# B&R Automation Studio project TrakFramework
Automation Studio 4.11.1.147; technology packages: mapp 5.18.0, mappFramework 1.0.0, mappMotion 5.18.0, mappView 5.18.0

## Configuration Config1

CPU PC_any, AutomationRuntime B4.92, Build 4.1.2, Safety 0.0, Vc V4.72.0

### Task classes (Cpu.sw)
```
Cyclic#1 (cycle 400 us, tolerance 0 us):
  AssemblyCt <- Source.AssemblyCtrl.prg
Cyclic#2 (cycle 2400 us, tolerance 2400 us):
  Deciders <- Source.Stations.Deciders.prg
Cyclic#3 (cycle 24000 us, tolerance 48000 us):
  Main <- Source.Main.prg
Cyclic#8 (cycle 800 us):
  Vis <- Source.Vis.Vis.prg
DataObjects: McAcpSys
NcDataObjects: McDriveLog
Binaries: mvLoader, FWRules, McAcpDrv, arsvcreg, McAcpSim, udbdef, TCData, arflatprv, arcoal, Config_3, arconfig, User, Role, sysconf, iomap, asfw, ashwac, ashwd, Config_2, Config_1, Config_4
Libraries: McBase, McAxis, McAcpTrak, standard, AsBrStr, TrakHelper, MpBase, ProcLogic, powerlnk, astime, arssl, fileio, runtime, asieccon, sys_lib
```

### Hardware
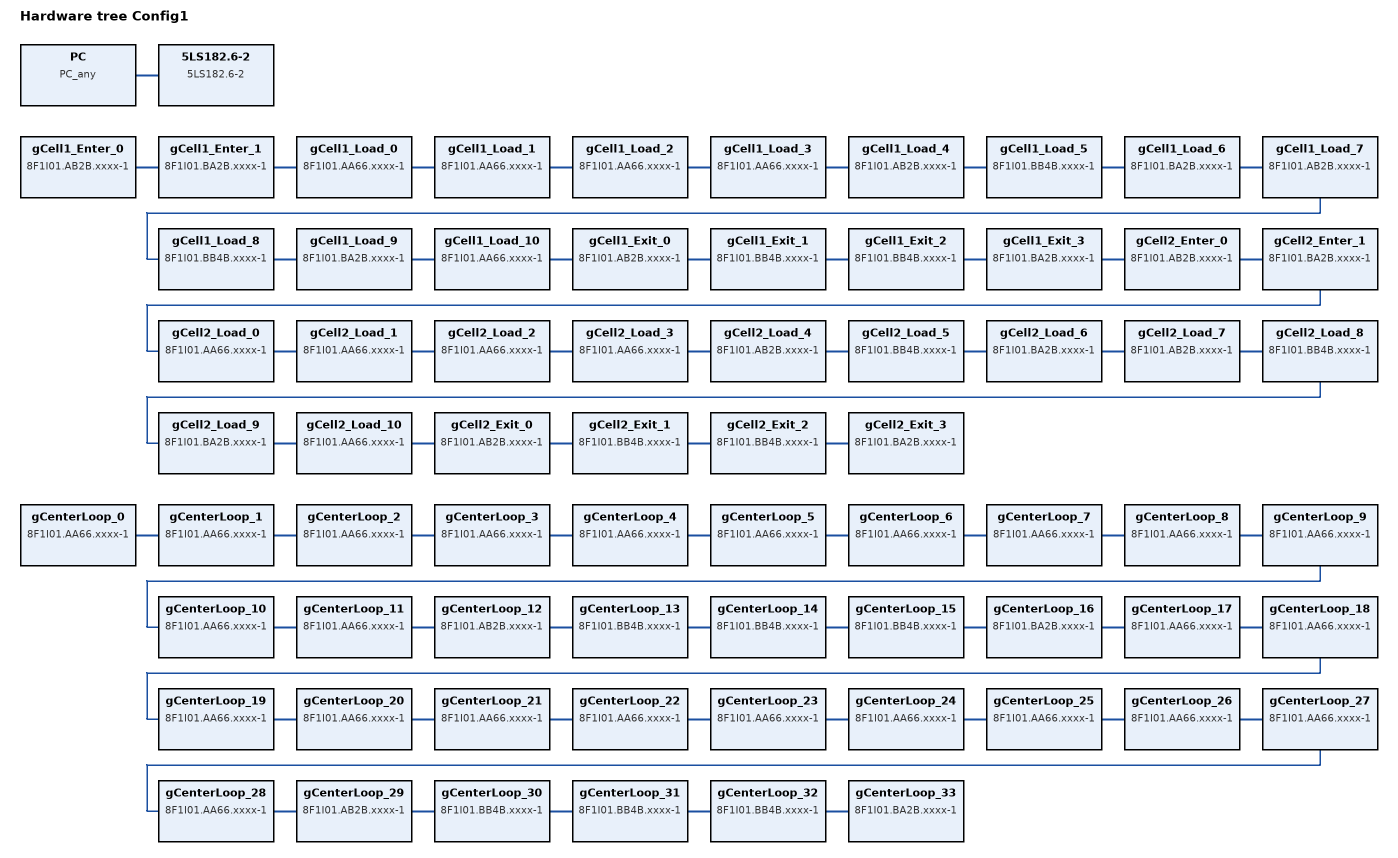
```
5LS182.6-2 : 5LS182.6-2 v1.9.0.0  [SL -> PC.SL1]
  Connector IF1:
    DNAConfiguration = manual
PC : PC_any v1.1.1.0 (OrderNumber=PC)
  ConfigurationID = BundlingSim_Config1
  SystemTick = 400
  Cyclic1Duration = 400
  Cyclic1Tolerance = 0
  Cyclic2Duration = 2400
  Cyclic2Tolerance = 2400
  Cyclic3Duration = 24000
  Cyclic3Tolerance = 48000
  Cyclic8Duration = 800
  FileDevice1
  FileDeviceName1 = SvgData
  FileDevicePath1 = ../../../../Logical/Scene
  ActivateOpcUa = 1
  OpcUaInformationModels_PV_Version = 1
gCell1_Enter_0 : 8F1I01.AB2B.xxxx-1 v1.0.0.2  [PLK1 -> gCenterLoop_33.PLK2 [Cable Type=PowerlinkCable, Length=10, Version=1.0.0.3]; PLK2 -> gCell1_Enter_1.PLK1 [Cable Type=PowerlinkCable, Length=10, Version=1.0.0.3]]
  DriveConfiguration:
    McTypeID = LLMConfig
  DriveConfiguration/Segment:
    Shape = STRAIGHT105_TO_CIRCULAR
    SegmentReference = gCell1_Enter_0
    StopReaction = UseAssemblySetting
    SpeedFilter = UseAssemblySetting
gCell1_Enter_1 : 8F1I01.BA2B.xxxx-1 v1.0.0.2  [PLK1 -> gCell1_Enter_0.PLK2 [Cable Type=PowerlinkCable, Length=10, Version=1.0.0.3]; PLK2 -> gCell1_Load_0.PLK1 [Cable Type=PowerlinkCable, Length=10, Version=1.0.0.3]]
  DriveConfiguration:
    McTypeID = LLMConfig
  DriveConfiguration/Segment:
    Shape = CIRCULAR_TO_STRAIGHT105
    SegmentReference = gCell1_Enter_1
    StopReaction = UseAssemblySetting
    SpeedFilter = UseAssemblySetting
gCell1_Exit_0 : 8F1I01.AB2B.xxxx-1 v1.0.0.2  [PLK1 -> gCell1_Load_10.PLK2 [Cable Type=PowerlinkCable, Length=10, Version=1.0.0.3]; PLK2 -> gCell1_Exit_1.PLK1 [Cable Type=PowerlinkCable, Length=10, Version=1.0.0.3]]
  DriveConfiguration:
    McTypeID = LLMConfig
  DriveConfiguration/Segment:
    Shape = STRAIGHT105_TO_CIRCULAR
    SegmentReference = gCell1_Exit_0
    StopReaction = UseAssemblySetting
    SpeedFilter = UseAssemblySetting
gCell1_Exit_1 : 8F1I01.BB4B.xxxx-1 v1.0.0.2  [PLK1 -> gCell1_Exit_0.PLK2 [Cable Type=PowerlinkCable, Length=10, Version=1.0.0.3]; PLK2 -> gCell1_Exit_2.PLK1 [Cable Type=PowerlinkCable, Length=10, Version=1.0.0.3]]
  DriveConfiguration:
    McTypeID = LLMConfig
  DriveConfiguration/Segment:
    Shape = CIRCULAR
    SegmentReference = gCell1_Exit_1
    StopReaction = UseAssemblySetting
    SpeedFilter = UseAssemblySetting
gCell1_Exit_2 : 8F1I01.BB4B.xxxx-1 v1.0.0.2  [PLK1 -> gCell1_Exit_1.PLK2 [Cable Type=PowerlinkCable, Length=10, Version=1.0.0.3]; PLK2 -> gCell1_Exit_3.PLK1 [Cable Type=PowerlinkCable, Length=10, Version=1.0.0.3]]
  DriveConfiguration:
    McTypeID = LLMConfig
  DriveConfiguration/Segment:
    Shape = CIRCULAR
    SegmentReference = gCell1_Exit_2
    StopReaction = UseAssemblySetting
    SpeedFilter = UseAssemblySetting
gCell1_Exit_3 : 8F1I01.BA2B.xxxx-1 v1.0.0.2  [PLK1 -> gCell1_Exit_2.PLK2 [Cable Type=PowerlinkCable, Length=10, Version=1.0.0.3]; PLK2 -> gCell2_Enter_0.PLK1 [Cable Type=PowerlinkCable, Length=10, Version=1.0.0.3]]
  DriveConfiguration:
    McTypeID = LLMConfig
  DriveConfiguration/Segment:
    Shape = CIRCULAR_TO_STRAIGHT105
    SegmentReference = gCell1_Exit_3
    StopReaction = UseAssemblySetting
    SpeedFilter = UseAssemblySetting
gCell1_Load_0 : 8F1I01.AA66.xxxx-1 v1.0.0.2  [PLK1 -> gCell1_Enter_1.PLK2 [Cable Type=PowerlinkCable, Length=10, Version=1.0.0.3]; PLK2 -> gCell1_Load_1.PLK1 [Cable Type=PowerlinkCable, Length=10, Version=1.0.0.3]]
  DriveConfiguration:
    McTypeID = LLMConfig
  DriveConfiguration/Segment:
    Shape = STRAIGHT660
    SegmentReference = gCell1_Load_0
    StopReaction = UseAssemblySetting
    SpeedFilter = UseAssemblySetting
gCell1_Load_1 : 8F1I01.AA66.xxxx-1 v1.0.0.2  [PLK1 -> gCell1_Load_0.PLK2 [Cable Type=PowerlinkCable, Length=10, Version=1.0.0.3]; PLK2 -> gCell1_Load_2.PLK1 [Cable Type=PowerlinkCable, Length=10, Version=1.0.0.3]]
  DriveConfiguration:
    McTypeID = LLMConfig
  DriveConfiguration/Segment:
    Shape = STRAIGHT660
    SegmentReference = gCell1_Load_1
    StopReaction = UseAssemblySetting
    SpeedFilter = UseAssemblySetting
gCell1_Load_10 : 8F1I01.AA66.xxxx-1 v1.0.0.2  [PLK1 -> gCell1_Load_9.PLK2 [Cable Type=PowerlinkCable, Length=10, Version=1.0.0.3]; PLK2 -> gCell1_Exit_0.PLK1 [Cable Type=PowerlinkCable, Length=10, Version=1.0.0.3]]
  DriveConfiguration:
    McTypeID = LLMConfig
  DriveConfiguration/Segment:
    Shape = STRAIGHT660
    SegmentReference = gCell1_Load_10
    StopReaction = UseAssemblySetting
    SpeedFilter = UseAssemblySetting
gCell1_Load_2 : 8F1I01.AA66.xxxx-1 v1.0.0.2  [PLK1 -> gCell1_Load_1.PLK2 [Cable Type=PowerlinkCable, Length=10, Version=1.0.0.3]; PLK2 -> gCell1_Load_3.PLK1 [Cable Type=PowerlinkCable, Length=10, Version=1.0.0.3]]
  DriveConfiguration:
    McTypeID = LLMConfig
  DriveConfiguration/Segment:
    Shape = STRAIGHT660
    SegmentReference = gCell1_Load_2
    StopReaction = UseAssemblySetting
    SpeedFilter = UseAssemblySetting
gCell1_Load_3 : 8F1I01.AA66.xxxx-1 v1.0.0.2  [PLK1 -> gCell1_Load_2.PLK2 [Cable Type=PowerlinkCable, Length=10, Version=1.0.0.3]; PLK2 -> gCell1_Load_4.PLK1 [Cable Type=PowerlinkCable, Length=10, Version=1.0.0.3]]
  DriveConfiguration:
    McTypeID = LLMConfig
  DriveConfiguration/Segment:
    Shape = STRAIGHT660
    SegmentReference = gCell1_Load_3
    StopReaction = UseAssemblySetting
    SpeedFilter = UseAssemblySetting
gCell1_Load_4 : 8F1I01.AB2B.xxxx-1 v1.0.0.2  [PLK1 -> gCell1_Load_3.PLK2 [Cable Type=PowerlinkCable, Length=10, Version=1.0.0.3]; PLK2 -> gCell1_Load_5.PLK1 [Cable Type=PowerlinkCable, Length=10, Version=1.0.0.3]]
  DriveConfiguration:
    McTypeID = LLMConfig
  DriveConfiguration/Segment:
    Shape = STRAIGHT105_TO_CIRCULAR
    SegmentReference = gCell1_Load_4
    StopReaction = UseAssemblySetting
    SpeedFilter = UseAssemblySetting
gCell1_Load_5 : 8F1I01.BB4B.xxxx-1 v1.0.0.2  [PLK1 -> gCell1_Load_4.PLK2 [Cable Type=PowerlinkCable, Length=10, Version=1.0.0.3]; PLK2 -> gCell1_Load_6.PLK1 [Cable Type=PowerlinkCable, Length=10, Version=1.0.0.3]]
  DriveConfiguration:
    McTypeID = LLMConfig
  DriveConfiguration/Segment:
    Shape = CIRCULAR
    SegmentReference = gCell1_Load_5
    StopReaction = UseAssemblySetting
    SpeedFilter = UseAssemblySetting
gCell1_Load_6 : 8F1I01.BA2B.xxxx-1 v1.0.0.2  [PLK1 -> gCell1_Load_5.PLK2 [Cable Type=PowerlinkCable, Length=10, Version=1.0.0.3]; PLK2 -> gCell1_Load_7.PLK1 [Cable Type=PowerlinkCable, Length=10, Version=1.0.0.3]]
  DriveConfiguration:
    McTypeID = LLMConfig
  DriveConfiguration/Segment:
    Shape = CIRCULAR_TO_STRAIGHT105
    SegmentReference = gCell1_Load_6
    StopReaction = UseAssemblySetting
    SpeedFilter = UseAssemblySetting
gCell1_Load_7 : 8F1I01.AB2B.xxxx-1 v1.0.0.2  [PLK1 -> gCell1_Load_6.PLK2 [Cable Type=PowerlinkCable, Length=10, Version=1.0.0.3]; PLK2 -> gCell1_Load_8.PLK1 [Cable Type=PowerlinkCable, Length=10, Version=1.0.0.3]]
  DriveConfiguration:
    McTypeID = LLMConfig
  DriveConfiguration/Segment:
    Shape = STRAIGHT105_TO_CIRCULAR
    SegmentReference = gCell1_Load_7
    StopReaction = UseAssemblySetting
    SpeedFilter = UseAssemblySetting
gCell1_Load_8 : 8F1I01.BB4B.xxxx-1 v1.0.0.2  [PLK1 -> gCell1_Load_7.PLK2 [Cable Type=PowerlinkCable, Length=10, Version=1.0.0.3]; PLK2 -> gCell1_Load_9.PLK1 [Cable Type=PowerlinkCable, Length=10, Version=1.0.0.3]]
  DriveConfiguration:
    McTypeID = LLMConfig
  DriveConfiguration/Segment:
    Shape = CIRCULAR
    SegmentReference = gCell1_Load_8
    StopReaction = UseAssemblySetting
    SpeedFilter = UseAssemblySetting
gCell1_Load_9 : 8F1I01.BA2B.xxxx-1 v1.0.0.2  [PLK1 -> gCell1_Load_8.PLK2 [Cable Type=PowerlinkCable, Length=10, Version=1.0.0.3]; PLK2 -> gCell1_Load_10.PLK1 [Cable Type=PowerlinkCable, Length=10, Version=1.0.0.3]]
  DriveConfiguration:
    McTypeID = LLMConfig
  DriveConfiguration/Segment:
    Shape = CIRCULAR_TO_STRAIGHT105
    SegmentReference = gCell1_Load_9
    StopReaction = UseAssemblySetting
    SpeedFilter = UseAssemblySetting
gCell2_Enter_0 : 8F1I01.AB2B.xxxx-1 v1.0.0.2  [PLK1 -> gCell1_Exit_3.PLK2 [Cable Type=PowerlinkCable, Length=10, Version=1.0.0.3]; PLK2 -> gCell2_Enter_1.PLK1 [Cable Type=PowerlinkCable, Length=10, Version=1.0.0.3]]
  DriveConfiguration:
    McTypeID = LLMConfig
  DriveConfiguration/Segment:
    Shape = STRAIGHT105_TO_CIRCULAR
    SegmentReference = gCell2_Enter_0
    StopReaction = UseAssemblySetting
    SpeedFilter = UseAssemblySetting
gCell2_Enter_1 : 8F1I01.BA2B.xxxx-1 v1.0.0.2  [PLK1 -> gCell2_Enter_0.PLK2 [Cable Type=PowerlinkCable, Length=10, Version=1.0.0.3]; PLK2 -> gCell2_Load_0.PLK1 [Cable Type=PowerlinkCable, Length=10, Version=1.0.0.3]]
  DriveConfiguration:
    McTypeID = LLMConfig
  DriveConfiguration/Segment:
    Shape = CIRCULAR_TO_STRAIGHT105
    SegmentReference = gCell2_Enter_1
    StopReaction = UseAssemblySetting
    SpeedFilter = UseAssemblySetting
gCell2_Exit_0 : 8F1I01.AB2B.xxxx-1 v1.0.0.2  [PLK1 -> gCell2_Load_10.PLK2 [Cable Type=PowerlinkCable, Length=10, Version=1.0.0.3]; PLK2 -> gCell2_Exit_1.PLK1 [Cable Type=PowerlinkCable, Length=10, Version=1.0.0.3]]
  DriveConfiguration:
    McTypeID = LLMConfig
  DriveConfiguration/Segment:
    Shape = STRAIGHT105_TO_CIRCULAR
    SegmentReference = gCell2_Exit_0
    StopReaction = UseAssemblySetting
    SpeedFilter = UseAssemblySetting
gCell2_Exit_1 : 8F1I01.BB4B.xxxx-1 v1.0.0.2  [PLK1 -> gCell2_Exit_0.PLK2 [Cable Type=PowerlinkCable, Length=10, Version=1.0.0.3]; PLK2 -> gCell2_Exit_2.PLK1 [Cable Type=PowerlinkCable, Length=10, Version=1.0.0.3]]
  DriveConfiguration:
    McTypeID = LLMConfig
  DriveConfiguration/Segment:
    Shape = CIRCULAR
    SegmentReference = gCell2_Exit_1
    StopReaction = UseAssemblySetting
    SpeedFilter = UseAssemblySetting
gCell2_Exit_2 : 8F1I01.BB4B.xxxx-1 v1.0.0.2  [PLK1 -> gCell2_Exit_1.PLK2 [Cable Type=PowerlinkCable, Length=10, Version=1.0.0.3]; PLK2 -> gCell2_Exit_3.PLK1 [Cable Type=PowerlinkCable, Length=10, Version=1.0.0.3]]
  DriveConfiguration:
    McTypeID = LLMConfig
  DriveConfiguration/Segment:
    Shape = CIRCULAR
    SegmentReference = gCell2_Exit_2
    StopReaction = UseAssemblySetting
    SpeedFilter = UseAssemblySetting
gCell2_Exit_3 : 8F1I01.BA2B.xxxx-1 v1.0.0.2  [PLK1 -> gCell2_Exit_2.PLK2 [Cable Type=PowerlinkCable, Length=10, Version=1.0.0.3]]
  DriveConfiguration:
    McTypeID = LLMConfig
  DriveConfiguration/Segment:
    Shape = CIRCULAR_TO_STRAIGHT105
    SegmentReference = gCell2_Exit_3
    StopReaction = UseAssemblySetting
    SpeedFilter = UseAssemblySetting
gCell2_Load_0 : 8F1I01.AA66.xxxx-1 v1.0.0.2  [PLK1 -> gCell2_Enter_1.PLK2 [Cable Type=PowerlinkCable, Length=10, Version=1.0.0.3]; PLK2 -> gCell2_Load_1.PLK1 [Cable Type=PowerlinkCable, Length=10, Version=1.0.0.3]]
  DriveConfiguration:
    McTypeID = LLMConfig
  DriveConfiguration/Segment:
    Shape = STRAIGHT660
    SegmentReference = gCell2_Load_0
    StopReaction = UseAssemblySetting
    SpeedFilter = UseAssemblySetting
gCell2_Load_1 : 8F1I01.AA66.xxxx-1 v1.0.0.2  [PLK1 -> gCell2_Load_0.PLK2 [Cable Type=PowerlinkCable, Length=10, Version=1.0.0.3]; PLK2 -> gCell2_Load_2.PLK1 [Cable Type=PowerlinkCable, Length=10, Version=1.0.0.3]]
  DriveConfiguration:
    McTypeID = LLMConfig
  DriveConfiguration/Segment:
    Shape = STRAIGHT660
    SegmentReference = gCell2_Load_1
    StopReaction = UseAssemblySetting
    SpeedFilter = UseAssemblySetting
gCell2_Load_10 : 8F1I01.AA66.xxxx-1 v1.0.0.2  [PLK1 -> gCell2_Load_9.PLK2 [Cable Type=PowerlinkCable, Length=10, Version=1.0.0.3]; PLK2 -> gCell2_Exit_0.PLK1 [Cable Type=PowerlinkCable, Length=10, Version=1.0.0.3]]
  DriveConfiguration:
    McTypeID = LLMConfig
  DriveConfiguration/Segment:
    Shape = STRAIGHT660
    SegmentReference = gCell2_Load_10
    StopReaction = UseAssemblySetting
    SpeedFilter = UseAssemblySetting
gCell2_Load_2 : 8F1I01.AA66.xxxx-1 v1.0.0.2  [PLK1 -> gCell2_Load_1.PLK2 [Cable Type=PowerlinkCable, Length=10, Version=1.0.0.3]; PLK2 -> gCell2_Load_3.PLK1 [Cable Type=PowerlinkCable, Length=10, Version=1.0.0.3]]
  DriveConfiguration:
    McTypeID = LLMConfig
  DriveConfiguration/Segment:
    Shape = STRAIGHT660
    SegmentReference = gCell2_Load_2
    StopReaction = UseAssemblySetting
    SpeedFilter = UseAssemblySetting
gCell2_Load_3 : 8F1I01.AA66.xxxx-1 v1.0.0.2  [PLK1 -> gCell2_Load_2.PLK2 [Cable Type=PowerlinkCable, Length=10, Version=1.0.0.3]; PLK2 -> gCell2_Load_4.PLK1 [Cable Type=PowerlinkCable, Length=10, Version=1.0.0.3]]
  DriveConfiguration:
    McTypeID = LLMConfig
  DriveConfiguration/Segment:
    Shape = STRAIGHT660
    SegmentReference = gCell2_Load_3
    StopReaction = UseAssemblySetting
    SpeedFilter = UseAssemblySetting
gCell2_Load_4 : 8F1I01.AB2B.xxxx-1 v1.0.0.2  [PLK1 -> gCell2_Load_3.PLK2 [Cable Type=PowerlinkCable, Length=10, Version=1.0.0.3]; PLK2 -> gCell2_Load_5.PLK1 [Cable Type=PowerlinkCable, Length=10, Version=1.0.0.3]]
  DriveConfiguration:
    McTypeID = LLMConfig
  DriveConfiguration/Segment:
    Shape = STRAIGHT105_TO_CIRCULAR
    SegmentReference = gCell2_Load_4
    StopReaction = UseAssemblySetting
    SpeedFilter = UseAssemblySetting
gCell2_Load_5 : 8F1I01.BB4B.xxxx-1 v1.0.0.2  [PLK1 -> gCell2_Load_4.PLK2 [Cable Type=PowerlinkCable, Length=10, Version=1.0.0.3]; PLK2 -> gCell2_Load_6.PLK1 [Cable Type=PowerlinkCable, Length=10, Version=1.0.0.3]]
  DriveConfiguration:
    McTypeID = LLMConfig
  DriveConfiguration/Segment:
    Shape = CIRCULAR
    SegmentReference = gCell2_Load_5
    StopReaction = UseAssemblySetting
    SpeedFilter = UseAssemblySetting
gCell2_Load_6 : 8F1I01.BA2B.xxxx-1 v1.0.0.2  [PLK1 -> gCell2_Load_5.PLK2 [Cable Type=PowerlinkCable, Length=10, Version=1.0.0.3]; PLK2 -> gCell2_Load_7.PLK1 [Cable Type=PowerlinkCable, Length=10, Version=1.0.0.3]]
  DriveConfiguration:
    McTypeID = LLMConfig
  DriveConfiguration/Segment:
    Shape = CIRCULAR_TO_STRAIGHT105
    SegmentReference = gCell2_Load_6
    StopReaction = UseAssemblySetting
    SpeedFilter = UseAssemblySetting
gCell2_Load_7 : 8F1I01.AB2B.xxxx-1 v1.0.0.2  [PLK1 -> gCell2_Load_6.PLK2 [Cable Type=PowerlinkCable, Length=10, Version=1.0.0.3]; PLK2 -> gCell2_Load_8.PLK1 [Cable Type=PowerlinkCable, Length=10, Version=1.0.0.3]]
  DriveConfiguration:
    McTypeID = LLMConfig
  DriveConfiguration/Segment:
    Shape = STRAIGHT105_TO_CIRCULAR
    SegmentReference = gCell2_Load_7
    StopReaction = UseAssemblySetting
    SpeedFilter = UseAssemblySetting
gCell2_Load_8 : 8F1I01.BB4B.xxxx-1 v1.0.0.2  [PLK1 -> gCell2_Load_7.PLK2 [Cable Type=PowerlinkCable, Length=10, Version=1.0.0.3]; PLK2 -> gCell2_Load_9.PLK1 [Cable Type=PowerlinkCable, Length=10, Version=1.0.0.3]]
  DriveConfiguration:
    McTypeID = LLMConfig
  DriveConfiguration/Segment:
    Shape = CIRCULAR
    SegmentReference = gCell2_Load_8
    StopReaction = UseAssemblySetting
    SpeedFilter = UseAssemblySetting
gCell2_Load_9 : 8F1I01.BA2B.xxxx-1 v1.0.0.2  [PLK1 -> gCell2_Load_8.PLK2 [Cable Type=PowerlinkCable, Length=10, Version=1.0.0.3]; PLK2 -> gCell2_Load_10.PLK1 [Cable Type=PowerlinkCable, Length=10, Version=1.0.0.3]]
  DriveConfiguration:
    McTypeID = LLMConfig
  DriveConfiguration/Segment:
    Shape = CIRCULAR_TO_STRAIGHT105
    SegmentReference = gCell2_Load_9
    StopReaction = UseAssemblySetting
    SpeedFilter = UseAssemblySetting
gCenterLoop_0 : 8F1I01.AA66.xxxx-1 v1.0.0.2  [PLK2 -> gCenterLoop_1.PLK1 [Cable Type=PowerlinkCable, Length=10, Version=1.0.0.3]; PLK3 -> 5LS182.6-2.IF1 [Cable Type=PowerlinkCable, Length=10, Version=1.0.0.3]]
  DriveConfiguration:
    McTypeID = LLMConfig
  DriveConfiguration/Segment:
    Shape = STRAIGHT660
    SegmentReference = gCenterLoop_0
    StopReaction = UseAssemblySetting
    SpeedFilter = UseAssemblySetting
gCenterLoop_1 : 8F1I01.AA66.xxxx-1 v1.0.0.2  [PLK1 -> gCenterLoop_0.PLK2 [Cable Type=PowerlinkCable, Length=10, Version=1.0.0.3]; PLK2 -> gCenterLoop_2.PLK1 [Cable Type=PowerlinkCable, Length=10, Version=1.0.0.3]]
  DriveConfiguration:
    McTypeID = LLMConfig
  DriveConfiguration/Segment:
    Shape = STRAIGHT660
    SegmentReference = gCenterLoop_1
    StopReaction = UseAssemblySetting
    SpeedFilter = UseAssemblySetting
gCenterLoop_10 : 8F1I01.AA66.xxxx-1 v1.0.0.2  [PLK1 -> gCenterLoop_9.PLK2 [Cable Type=PowerlinkCable, Length=10, Version=1.0.0.3]; PLK2 -> gCenterLoop_11.PLK1 [Cable Type=PowerlinkCable, Length=10, Version=1.0.0.3]]
  DriveConfiguration:
    McTypeID = LLMConfig
  DriveConfiguration/Segment:
    Shape = STRAIGHT660
    SegmentReference = gCenterLoop_10
    StopReaction = UseAssemblySetting
    SpeedFilter = UseAssemblySetting
gCenterLoop_11 : 8F1I01.AA66.xxxx-1 v1.0.0.2  [PLK1 -> gCenterLoop_10.PLK2 [Cable Type=PowerlinkCable, Length=10, Version=1.0.0.3]; PLK2 -> gCenterLoop_12.PLK1 [Cable Type=PowerlinkCable, Length=10, Version=1.0.0.3]]
  DriveConfiguration:
    McTypeID = LLMConfig
  DriveConfiguration/Segment:
    Shape = STRAIGHT660
    SegmentReference = gCenterLoop_11
    StopReaction = UseAssemblySetting
    SpeedFilter = UseAssemblySetting
gCenterLoop_12 : 8F1I01.AB2B.xxxx-1 v1.0.0.2  [PLK1 -> gCenterLoop_11.PLK2 [Cable Type=PowerlinkCable, Length=10, Version=1.0.0.3]; PLK2 -> gCenterLoop_13.PLK1 [Cable Type=PowerlinkCable, Length=10, Version=1.0.0.3]]
  DriveConfiguration:
    McTypeID = LLMConfig
  DriveConfiguration/Segment:
    Shape = STRAIGHT105_TO_CIRCULAR
    SegmentReference = gCenterLoop_12
    StopReaction = UseAssemblySetting
    SpeedFilter = UseAssemblySetting
gCenterLoop_13 : 8F1I01.BB4B.xxxx-1 v1.0.0.2  [PLK1 -> gCenterLoop_12.PLK2 [Cable Type=PowerlinkCable, Length=10, Version=1.0.0.3]; PLK2 -> gCenterLoop_14.PLK1 [Cable Type=PowerlinkCable, Length=10, Version=1.0.0.3]]
  DriveConfiguration:
    McTypeID = LLMConfig
  DriveConfiguration/Segment:
    Shape = CIRCULAR
    SegmentReference = gCenterLoop_13
    StopReaction = UseAssemblySetting
    SpeedFilter = UseAssemblySetting
gCenterLoop_14 : 8F1I01.BB4B.xxxx-1 v1.0.0.2  [PLK1 -> gCenterLoop_13.PLK2 [Cable Type=PowerlinkCable, Length=10, Version=1.0.0.3]; PLK2 -> gCenterLoop_15.PLK1 [Cable Type=PowerlinkCable, Length=10, Version=1.0.0.3]]
  DriveConfiguration:
    McTypeID = LLMConfig
  DriveConfiguration/Segment:
    Shape = CIRCULAR
    SegmentReference = gCenterLoop_14
    StopReaction = UseAssemblySetting
    SpeedFilter = UseAssemblySetting
gCenterLoop_15 : 8F1I01.BB4B.xxxx-1 v1.0.0.2  [PLK1 -> gCenterLoop_14.PLK2 [Cable Type=PowerlinkCable, Length=10, Version=1.0.0.3]; PLK2 -> gCenterLoop_16.PLK1 [Cable Type=PowerlinkCable, Length=10, Version=1.0.0.3]]
  DriveConfiguration:
    McTypeID = LLMConfig
  DriveConfiguration/Segment:
    Shape = CIRCULAR
    SegmentReference = gCenterLoop_15
    StopReaction = UseAssemblySetting
    SpeedFilter = UseAssemblySetting
gCenterLoop_16 : 8F1I01.BA2B.xxxx-1 v1.0.0.2  [PLK1 -> gCenterLoop_15.PLK2 [Cable Type=PowerlinkCable, Length=10, Version=1.0.0.3]; PLK2 -> gCenterLoop_17.PLK1 [Cable Type=PowerlinkCable, Length=10, Version=1.0.0.3]]
  DriveConfiguration:
    McTypeID = LLMConfig
  DriveConfiguration/Segment:
    Shape = CIRCULAR_TO_STRAIGHT105
    SegmentReference = gCenterLoop_16
    StopReaction = UseAssemblySetting
    SpeedFilter = UseAssemblySetting
gCenterLoop_17 : 8F1I01.AA66.xxxx-1 v1.0.0.2  [PLK1 -> gCenterLoop_16.PLK2 [Cable Type=PowerlinkCable, Length=10, Version=1.0.0.3]; PLK2 -> gCenterLoop_18.PLK1 [Cable Type=PowerlinkCable, Length=10, Version=1.0.0.3]]
  DriveConfiguration:
    McTypeID = LLMConfig
  DriveConfiguration/Segment:
    Shape = STRAIGHT660
    SegmentReference = gCenterLoop_17
    StopReaction = UseAssemblySetting
    SpeedFilter = UseAssemblySetting
gCenterLoop_18 : 8F1I01.AA66.xxxx-1 v1.0.0.2  [PLK1 -> gCenterLoop_17.PLK2 [Cable Type=PowerlinkCable, Length=10, Version=1.0.0.3]; PLK2 -> gCenterLoop_19.PLK1 [Cable Type=PowerlinkCable, Length=10, Version=1.0.0.3]]
  DriveConfiguration:
    McTypeID = LLMConfig
  DriveConfiguration/Segment:
    Shape = STRAIGHT660
    SegmentReference = gCenterLoop_18
    StopReaction = UseAssemblySetting
    SpeedFilter = UseAssemblySetting
gCenterLoop_19 : 8F1I01.AA66.xxxx-1 v1.0.0.2  [PLK1 -> gCenterLoop_18.PLK2 [Cable Type=PowerlinkCable, Length=10, Version=1.0.0.3]; PLK2 -> gCenterLoop_20.PLK1 [Cable Type=PowerlinkCable, Length=10, Version=1.0.0.3]]
  DriveConfiguration:
    McTypeID = LLMConfig
  DriveConfiguration/Segment:
    Shape = STRAIGHT660
    SegmentReference = gCenterLoop_19
    StopReaction = UseAssemblySetting
    SpeedFilter = UseAssemblySetting
gCenterLoop_2 : 8F1I01.AA66.xxxx-1 v1.0.0.2  [PLK1 -> gCenterLoop_1.PLK2 [Cable Type=PowerlinkCable, Length=10, Version=1.0.0.3]; PLK2 -> gCenterLoop_3.PLK1 [Cable Type=PowerlinkCable, Length=10, Version=1.0.0.3]]
  DriveConfiguration:
    McTypeID = LLMConfig
  DriveConfiguration/Segment:
    Shape = STRAIGHT660
    SegmentReference = gCenterLoop_2
    StopReaction = UseAssemblySetting
    SpeedFilter = UseAssemblySetting
gCenterLoop_20 : 8F1I01.AA66.xxxx-1 v1.0.0.2  [PLK1 -> gCenterLoop_19.PLK2 [Cable Type=PowerlinkCable, Length=10, Version=1.0.0.3]; PLK2 -> gCenterLoop_21.PLK1 [Cable Type=PowerlinkCable, Length=10, Version=1.0.0.3]]
  DriveConfiguration:
    McTypeID = LLMConfig
  DriveConfiguration/Segment:
    Shape = STRAIGHT660
    SegmentReference = gCenterLoop_20
    StopReaction = UseAssemblySetting
    SpeedFilter = UseAssemblySetting
gCenterLoop_21 : 8F1I01.AA66.xxxx-1 v1.0.0.2  [PLK1 -> gCenterLoop_20.PLK2 [Cable Type=PowerlinkCable, Length=10, Version=1.0.0.3]; PLK2 -> gCenterLoop_22.PLK1 [Cable Type=PowerlinkCable, Length=10, Version=1.0.0.3]]
  DriveConfiguration:
    McTypeID = LLMConfig
  DriveConfiguration/Segment:
    Shape = STRAIGHT660
    SegmentReference = gCenterLoop_21
    StopReaction = UseAssemblySetting
    SpeedFilter = UseAssemblySetting
gCenterLoop_22 : 8F1I01.AA66.xxxx-1 v1.0.0.2  [PLK1 -> gCenterLoop_21.PLK2 [Cable Type=PowerlinkCable, Length=10, Version=1.0.0.3]; PLK2 -> gCenterLoop_23.PLK1 [Cable Type=PowerlinkCable, Length=10, Version=1.0.0.3]]
  DriveConfiguration:
    McTypeID = LLMConfig
  DriveConfiguration/Segment:
    Shape = STRAIGHT660
    SegmentReference = gCenterLoop_22
    StopReaction = UseAssemblySetting
    SpeedFilter = UseAssemblySetting
gCenterLoop_23 : 8F1I01.AA66.xxxx-1 v1.0.0.2  [PLK1 -> gCenterLoop_22.PLK2 [Cable Type=PowerlinkCable, Length=10, Version=1.0.0.3]; PLK2 -> gCenterLoop_24.PLK1 [Cable Type=PowerlinkCable, Length=10, Version=1.0.0.3]]
  DriveConfiguration:
    McTypeID = LLMConfig
  DriveConfiguration/Segment:
    Shape = STRAIGHT660
    SegmentReference = gCenterLoop_23
    StopReaction = UseAssemblySetting
    SpeedFilter = UseAssemblySetting
gCenterLoop_24 : 8F1I01.AA66.xxxx-1 v1.0.0.2  [PLK1 -> gCenterLoop_23.PLK2 [Cable Type=PowerlinkCable, Length=10, Version=1.0.0.3]; PLK2 -> gCenterLoop_25.PLK1 [Cable Type=PowerlinkCable, Length=10, Version=1.0.0.3]]
  DriveConfiguration:
    McTypeID = LLMConfig
  DriveConfiguration/Segment:
    Shape = STRAIGHT660
    SegmentReference = gCenterLoop_24
    StopReaction = UseAssemblySetting
    SpeedFilter = UseAssemblySetting
gCenterLoop_25 : 8F1I01.AA66.xxxx-1 v1.0.0.2  [PLK1 -> gCenterLoop_24.PLK2 [Cable Type=PowerlinkCable, Length=10, Version=1.0.0.3]; PLK2 -> gCenterLoop_26.PLK1 [Cable Type=PowerlinkCable, Length=10, Version=1.0.0.3]]
  DriveConfiguration:
    McTypeID = LLMConfig
  DriveConfiguration/Segment:
    Shape = STRAIGHT660
    SegmentReference = gCenterLoop_25
    StopReaction = UseAssemblySetting
    SpeedFilter = UseAssemblySetting
gCenterLoop_26 : 8F1I01.AA66.xxxx-1 v1.0.0.2  [PLK1 -> gCenterLoop_25.PLK2 (NodeNumber=27) [Cable Type=PowerlinkCable, Length=10, Version=1.0.0.3]; PLK2 -> gCenterLoop_27.PLK1 (NodeNumber=27) [Cable Type=PowerlinkCable, Length=10, Version=1.0.0.3]]
  DriveConfiguration:
    McTypeID = LLMConfig
  DriveConfiguration/Segment:
    Shape = STRAIGHT660
    SegmentReference = gCenterLoop_26
    StopReaction = UseAssemblySetting
    SpeedFilter = UseAssemblySetting
gCenterLoop_27 : 8F1I01.AA66.xxxx-1 v1.0.0.2  [PLK1 -> gCenterLoop_26.PLK2 [Cable Type=PowerlinkCable, Length=10, Version=1.0.0.3]; PLK2 -> gCenterLoop_28.PLK1 [Cable Type=PowerlinkCable, Length=10, Version=1.0.0.3]]
  DriveConfiguration:
    McTypeID = LLMConfig
  DriveConfiguration/Segment:
    Shape = STRAIGHT660
    SegmentReference = gCenterLoop_27
    StopReaction = UseAssemblySetting
    SpeedFilter = UseAssemblySetting
gCenterLoop_28 : 8F1I01.AA66.xxxx-1 v1.0.0.2  [PLK1 -> gCenterLoop_27.PLK2 [Cable Type=PowerlinkCable, Length=10, Version=1.0.0.3]; PLK2 -> gCenterLoop_29.PLK1 [Cable Type=PowerlinkCable, Length=10, Version=1.0.0.3]]
  DriveConfiguration:
    McTypeID = LLMConfig
  DriveConfiguration/Segment:
    Shape = STRAIGHT660
    SegmentReference = gCenterLoop_28
    StopReaction = UseAssemblySetting
    SpeedFilter = UseAssemblySetting
gCenterLoop_29 : 8F1I01.AB2B.xxxx-1 v1.0.0.2  [PLK1 -> gCenterLoop_28.PLK2 [Cable Type=PowerlinkCable, Length=10, Version=1.0.0.3]; PLK2 -> gCenterLoop_30.PLK1 [Cable Type=PowerlinkCable, Length=10, Version=1.0.0.3]]
  DriveConfiguration:
    McTypeID = LLMConfig
  DriveConfiguration/Segment:
    Shape = STRAIGHT105_TO_CIRCULAR
    SegmentReference = gCenterLoop_29
    StopReaction = UseAssemblySetting
    SpeedFilter = UseAssemblySetting
gCenterLoop_3 : 8F1I01.AA66.xxxx-1 v1.0.0.2  [PLK1 -> gCenterLoop_2.PLK2 [Cable Type=PowerlinkCable, Length=10, Version=1.0.0.3]; PLK2 -> gCenterLoop_4.PLK1 [Cable Type=PowerlinkCable, Length=10, Version=1.0.0.3]]
  DriveConfiguration:
    McTypeID = LLMConfig
  DriveConfiguration/Segment:
    Shape = STRAIGHT660
    SegmentReference = gCenterLoop_3
    StopReaction = UseAssemblySetting
    SpeedFilter = UseAssemblySetting
gCenterLoop_30 : 8F1I01.BB4B.xxxx-1 v1.0.0.2  [PLK1 -> gCenterLoop_29.PLK2 [Cable Type=PowerlinkCable, Length=10, Version=1.0.0.3]; PLK2 -> gCenterLoop_31.PLK1 [Cable Type=PowerlinkCable, Length=10, Version=1.0.0.3]]
  DriveConfiguration:
    McTypeID = LLMConfig
  DriveConfiguration/Segment:
    Shape = CIRCULAR
    SegmentReference = gCenterLoop_30
    StopReaction = UseAssemblySetting
    SpeedFilter = UseAssemblySetting
gCenterLoop_31 : 8F1I01.BB4B.xxxx-1 v1.0.0.2  [PLK1 -> gCenterLoop_30.PLK2 [Cable Type=PowerlinkCable, Length=10, Version=1.0.0.3]; PLK2 -> gCenterLoop_32.PLK1 [Cable Type=PowerlinkCable, Length=10, Version=1.0.0.3]]
  DriveConfiguration:
    McTypeID = LLMConfig
  DriveConfiguration/Segment:
    Shape = CIRCULAR
    SegmentReference = gCenterLoop_31
    StopReaction = UseAssemblySetting
    SpeedFilter = UseAssemblySetting
gCenterLoop_32 : 8F1I01.BB4B.xxxx-1 v1.0.0.2  [PLK1 -> gCenterLoop_31.PLK2 [Cable Type=PowerlinkCable, Length=10, Version=1.0.0.3]; PLK2 -> gCenterLoop_33.PLK1 [Cable Type=PowerlinkCable, Length=10, Version=1.0.0.3]]
  DriveConfiguration:
    McTypeID = LLMConfig
  DriveConfiguration/Segment:
    Shape = CIRCULAR
    SegmentReference = gCenterLoop_32
    StopReaction = UseAssemblySetting
    SpeedFilter = UseAssemblySetting
gCenterLoop_33 : 8F1I01.BA2B.xxxx-1 v1.0.0.2  [PLK1 -> gCenterLoop_32.PLK2 [Cable Type=PowerlinkCable, Length=10, Version=1.0.0.3]; PLK2 -> gCell1_Enter_0.PLK1 [Cable Type=PowerlinkCable, Length=10, Version=1.0.0.3]]
  DriveConfiguration:
    McTypeID = LLMConfig
  DriveConfiguration/Segment:
    Shape = CIRCULAR_TO_STRAIGHT105
    SegmentReference = gCenterLoop_33
    StopReaction = UseAssemblySetting
    SpeedFilter = UseAssemblySetting
gCenterLoop_4 : 8F1I01.AA66.xxxx-1 v1.0.0.2  [PLK1 -> gCenterLoop_3.PLK2 [Cable Type=PowerlinkCable, Length=10, Version=1.0.0.3]; PLK2 -> gCenterLoop_5.PLK1 [Cable Type=PowerlinkCable, Length=10, Version=1.0.0.3]]
  DriveConfiguration:
    McTypeID = LLMConfig
  DriveConfiguration/Segment:
    Shape = STRAIGHT660
    SegmentReference = gCenterLoop_4
    StopReaction = UseAssemblySetting
    SpeedFilter = UseAssemblySetting
gCenterLoop_5 : 8F1I01.AA66.xxxx-1 v1.0.0.2  [PLK1 -> gCenterLoop_4.PLK2 [Cable Type=PowerlinkCable, Length=10, Version=1.0.0.3]; PLK2 -> gCenterLoop_6.PLK1 [Cable Type=PowerlinkCable, Length=10, Version=1.0.0.3]]
  DriveConfiguration:
    McTypeID = LLMConfig
  DriveConfiguration/Segment:
    Shape = STRAIGHT660
    SegmentReference = gCenterLoop_5
    StopReaction = UseAssemblySetting
    SpeedFilter = UseAssemblySetting
gCenterLoop_6 : 8F1I01.AA66.xxxx-1 v1.0.0.2  [PLK1 -> gCenterLoop_5.PLK2 [Cable Type=PowerlinkCable, Length=10, Version=1.0.0.3]; PLK2 -> gCenterLoop_7.PLK1 [Cable Type=PowerlinkCable, Length=10, Version=1.0.0.3]]
  DriveConfiguration:
    McTypeID = LLMConfig
  DriveConfiguration/Segment:
    Shape = STRAIGHT660
    SegmentReference = gCenterLoop_6
    StopReaction = UseAssemblySetting
    SpeedFilter = UseAssemblySetting
gCenterLoop_7 : 8F1I01.AA66.xxxx-1 v1.0.0.2  [PLK1 -> gCenterLoop_6.PLK2 [Cable Type=PowerlinkCable, Length=10, Version=1.0.0.3]; PLK2 -> gCenterLoop_8.PLK1 [Cable Type=PowerlinkCable, Length=10, Version=1.0.0.3]]
  DriveConfiguration:
    McTypeID = LLMConfig
  DriveConfiguration/Segment:
    Shape = STRAIGHT660
    SegmentReference = gCenterLoop_7
    StopReaction = UseAssemblySetting
    SpeedFilter = UseAssemblySetting
gCenterLoop_8 : 8F1I01.AA66.xxxx-1 v1.0.0.2  [PLK1 -> gCenterLoop_7.PLK2 [Cable Type=PowerlinkCable, Length=10, Version=1.0.0.3]; PLK2 -> gCenterLoop_9.PLK1 [Cable Type=PowerlinkCable, Length=10, Version=1.0.0.3]]
  DriveConfiguration:
    McTypeID = LLMConfig
  DriveConfiguration/Segment:
    Shape = STRAIGHT660
    SegmentReference = gCenterLoop_8
    StopReaction = UseAssemblySetting
    SpeedFilter = UseAssemblySetting
gCenterLoop_9 : 8F1I01.AA66.xxxx-1 v1.0.0.2  [PLK1 -> gCenterLoop_8.PLK2 [Cable Type=PowerlinkCable, Length=10, Version=1.0.0.3]; PLK2 -> gCenterLoop_10.PLK1 [Cable Type=PowerlinkCable, Length=10, Version=1.0.0.3]]
  DriveConfiguration:
    McTypeID = LLMConfig
  DriveConfiguration/Segment:
    Shape = STRAIGHT660
    SegmentReference = gCenterLoop_9
    StopReaction = UseAssemblySetting
    SpeedFilter = UseAssemblySetting
```

### Config_1.assembly - PC/mappMotion/Config_1.assembly
```
Element gTestAssembly (Type=assembly)
  Tracks:
    TrackSeparation = 0.030
    Track[1]:
      Segments:
        SegmentRef[1] = ::gCenterLoop_0
        SegmentRef[2] = ::gCenterLoop_1
        SegmentRef[3] = ::gCenterLoop_2
        SegmentRef[4] = ::gCenterLoop_3
        SegmentRef[5] = ::gCenterLoop_4
        SegmentRef[6] = ::gCenterLoop_5
        SegmentRef[7] = ::gCenterLoop_6
        SegmentRef[8] = ::gCenterLoop_7
        SegmentRef[9] = ::gCenterLoop_8
        SegmentRef[10] = ::gCenterLoop_9
        SegmentRef[11] = ::gCenterLoop_10
        SegmentRef[12] = ::gCenterLoop_11
        SegmentRef[13] = ::gCenterLoop_12
        SegmentRef[14] = ::gCenterLoop_13
        SegmentRef[15] = ::gCenterLoop_14
        SegmentRef[16] = ::gCenterLoop_15
        SegmentRef[17] = ::gCenterLoop_16
        SegmentRef[18] = ::gCenterLoop_17
        SegmentRef[19] = ::gCenterLoop_18
        SegmentRef[20] = ::gCenterLoop_19
        SegmentRef[21] = ::gCenterLoop_20
        SegmentRef[22] = ::gCenterLoop_21
        SegmentRef[23] = ::gCenterLoop_22
        SegmentRef[24] = ::gCenterLoop_23
        SegmentRef[25] = ::gCenterLoop_24
        SegmentRef[26] = ::gCenterLoop_25
        SegmentRef[27] = ::gCenterLoop_26
        SegmentRef[28] = ::gCenterLoop_27
        SegmentRef[29] = ::gCenterLoop_28
        SegmentRef[30] = ::gCenterLoop_29
        SegmentRef[31] = ::gCenterLoop_30
        SegmentRef[32] = ::gCenterLoop_31
        SegmentRef[33] = ::gCenterLoop_32
        SegmentRef[34] = ::gCenterLoop_33
      Position = Absolute
        SegmentRef = ::gCenterLoop_0
        SegmentCountDirection = RightToLeft
        Translation:
          X = 0.0
          Y = 0.0
          Z = 0.0
        Orientation:
          Angle1 = 0.0
          Angle2 = 0.0
          Angle3 = 0.0
    Track[2]:
      Segments:
        SegmentRef[1] = ::gCell1_Enter_0
        SegmentRef[2] = ::gCell1_Enter_1
      Position = RelativeToOne
        TrackSegmentPosition:
          SegmentRef = ::gCell1_Enter_1
          PositionRelativeTo = FromEnd
        Base:
          SegmentRef = ::gCenterLoop_33
          Position = 0.09
          PositionRelativeTo = FromEnd
    Track[3]:
      Segments:
        SegmentRef[1] = ::gCell1_Load_0
        SegmentRef[2] = ::gCell1_Load_1
        SegmentRef[3] = ::gCell1_Load_2
        SegmentRef[4] = ::gCell1_Load_3
        SegmentRef[5] = ::gCell1_Load_4
        SegmentRef[6] = ::gCell1_Load_5
        SegmentRef[7] = ::gCell1_Load_6
        SegmentRef[8] = ::gCell1_Load_7
        SegmentRef[9] = ::gCell1_Load_8
        SegmentRef[10] = ::gCell1_Load_9
        SegmentRef[11] = ::gCell1_Load_10
      Position = RelativeToOne
        TrackSegmentPosition:
          SegmentRef = ::gCell1_Load_0
        Base:
          SegmentRef = ::gCell1_Enter_0
          Position = 0.09
    Track[4]:
      Segments:
        SegmentRef[1] = ::gCell1_Exit_0
        SegmentRef[2] = ::gCell1_Exit_1
        SegmentRef[3] = ::gCell1_Exit_2
        SegmentRef[4] = ::gCell1_Exit_3
      Position = RelativeToOne
        TrackSegmentPosition:
          SegmentRef = ::gCell1_Exit_3
          PositionRelativeTo = FromEnd
        Base:
          SegmentRef = ::gCell1_Load_10
          Position = 0.09
          PositionRelativeTo = FromEnd
    Track[5]:
      Segments:
        SegmentRef[1] = ::gCell2_Enter_0
        SegmentRef[2] = ::gCell2_Enter_1
      Position = RelativeToOne
        TrackSegmentPosition:
          SegmentRef = ::gCell2_Enter_1
          PositionRelativeTo = FromEnd
        Base:
          SegmentRef = ::gCenterLoop_6
          Position = 0.33
    Track[6]:
      Segments:
        SegmentRef[1] = ::gCell2_Load_0
        SegmentRef[2] = ::gCell2_Load_1
        SegmentRef[3] = ::gCell2_Load_2
        SegmentRef[4] = ::gCell2_Load_3
        SegmentRef[5] = ::gCell2_Load_4
        SegmentRef[6] = ::gCell2_Load_5
        SegmentRef[7] = ::gCell2_Load_6
        SegmentRef[8] = ::gCell2_Load_7
        SegmentRef[9] = ::gCell2_Load_8
        SegmentRef[10] = ::gCell2_Load_9
        SegmentRef[11] = ::gCell2_Load_10
      Position = RelativeToOne
        TrackSegmentPosition:
          SegmentRef = ::gCell2_Load_0
        Base:
          SegmentRef = ::gCell2_Enter_0
          Position = 0.09
    Track[7]:
      Segments:
        SegmentRef[1] = ::gCell2_Exit_0
        SegmentRef[2] = ::gCell2_Exit_1
        SegmentRef[3] = ::gCell2_Exit_2
        SegmentRef[4] = ::gCell2_Exit_3
      Position = RelativeToOne
        TrackSegmentPosition:
          SegmentRef = ::gCell2_Exit_3
          PositionRelativeTo = FromEnd
        Base:
          SegmentRef = ::gCell2_Load_10
          Position = 0.09
          PositionRelativeTo = FromEnd
  CommonSegmentSettings:
    SegmentSimulationOnPLC = Off
    ElongationCompensation = Inactive
    StopReaction = InductionHalt
    SpeedFilter = NotUsed
    ControllerParameters:
      DefaultParameter:
        Controller:
          Position:
            ProportionalGain = 0.0
          Speed:
            ProportionalGain = 0.0
            IntegrationTime = 0.0
          FeedForward:
            TotalMass = 0.0
            ForcePositive = 0.0
            ForceNegative = 0.0
            SpeedForceFactor = 0.0
            ForceLoad = 0.0
        MovementErrorLimits:
          PositionError = 0.0
          VelocityError = 0.0
      AdditionalParameterSets = NotUsed
    ScopeOfErrorReaction = Assembly
    ShuttleIdentificationTime = 0
  Shuttles:
    MaxShuttleCount = 100
    MaxShuttleCommandCount = 0
    UseConvoys = Inactive
    DistanceReserve:
      Collision = 0.002
      ErrorStop = 0.006
    ShuttleStereotypes:
      ShuttleStRef[1] = ShuttleStereotype_1
    MagnetPlateConfigurations:
      ShuttleType[1] = 8F1SA.100.xxxxxx-x
    CollisionAvoidance:
      Strategy = Constant
      MaximumModelDimensions:
        Length:
          ExtentToFront = 0.025
          ExtentToBack = 0.025
        Width:
          Width = 0.046
  Visualization:
    MonitoringPv = ::gShuttleMon
    ProcessingTaskClass = 1
```

### Config_2.shuttlestereotype - PC/mappMotion/Config_2.shuttlestereotype
```
Element ShuttleStereotype_1 (Type=shuttlestereotype)
  MeasurementUnit = 5067858
  MeasurementResolution = 0.00001
  MovementLimits = Internal
    VelocityIsReadOnly = 0
    Velocity:
      Velocity = 2
    AccelerationIsReadOnly = 0
    Acceleration:
      Acceleration = 20.0
    DecelerationIsReadOnly = 0
    Deceleration:
      Deceleration = 20.0
    UpdateMode = Immediately
  JerkFilter = Used
    JerkTime = 0.02
  UserData:
    Size = 28
```

### Config_3.sector - PC/mappMotion/Config_3.sector
```
Element secStartup (Type=sector)
  Type = Composed
    StartSegment:
      SegmentRef = ::gCenterLoop_21
    IntermediateSegments:
      SegmentRef[1] = ::gCenterLoop_22
      SegmentRef[2] = ::gCenterLoop_23
      SegmentRef[3] = ::gCenterLoop_24
      SegmentRef[4] = ::gCenterLoop_25
      SegmentRef[5] = ::gCenterLoop_26
      SegmentRef[6] = ::gCenterLoop_27
      SegmentRef[7] = ::gCenterLoop_28
      SegmentRef[8] = ::gCenterLoop_29
      SegmentRef[9] = ::gCenterLoop_30
      SegmentRef[10] = ::gCenterLoop_31
    EndSegment:
      SegmentRef = ::gCenterLoop_32
      PositionRelativeTo = FromEnd
  Alarms = None
Element secLoadDecision (Type=sector)
  Type = Composed
    StartSegment:
      SegmentRef = ::gCenterLoop_33
    EndSegment:
      SegmentRef = ::gCenterLoop_33
      PositionRelativeTo = FromEnd
  Alarms = None
Element secProcess1 (Type=sector)
  Type = Composed
    StartSegment:
      SegmentRef = ::gCell1_Load_2
    EndSegment:
      SegmentRef = ::gCell1_Load_2
      PositionRelativeTo = FromEnd
  Alarms = None
Element secProcess2 (Type=sector)
  Type = Composed
    StartSegment:
      SegmentRef = ::gCell2_Load_2
    EndSegment:
      SegmentRef = ::gCell2_Load_2
      PositionRelativeTo = FromEnd
  Alarms = None
```

### Config_4.processpointlist - PC/mappMotion/Config_4.processpointlist
```
Element ProcessPointList_1 (Type=processpointlist)
  ProcessPoint[0]:
    Name = ppLoadDecision
    SectorRef = secLoadDecision
    TriggerEventBufferSize = 10
    BarrierFunctionality = Off
  ProcessPoint[1]:
    Name = ppProcess1
    SectorRef = secProcess1
    Position = 0.00
    TriggerEventBufferSize = 10
    BarrierFunctionality = Off
  ProcessPoint[2]:
    Name = ppProcess2
    SectorRef = secProcess2
    Position = 0
    TriggerEventBufferSize = 10
    BarrierFunctionality = Off
```

## Logical view

Binary libraries used (declarations not repeated): operator, runtime, astime, AsIecCon, standard, AsBrStr, McBase, McAcpTrak 5.18.0, McAxis, MpBase

### Global.typ - Global data types
```iecst
(*Main Interfaces Types*)

TYPE
	MainIfTyp : 	STRUCT
		Cmd : MainIfCmdTyp;
		Par : MainIfParTyp;
		Sts : MainIfStsTyp;
	END_STRUCT;
	MainIfCmdTyp : 	STRUCT
		Power : BOOL;
		Run : BOOL;
		Reset : BOOL;
		ShowError : BOOL;
	END_STRUCT;
	MainIfParTyp : 	STRUCT
		DefaultVelocity : REAL;
		DefaultAccel : REAL;
		DefaultDecel : REAL;
	END_STRUCT;
	MainIfStsTyp : 	STRUCT
		TrakPowered : BOOL;
		Running : BOOL;
		Error : BOOL;
	END_STRUCT;
END_TYPE

(*Trak Assembly Interface Types*)

TYPE
	AcpTrakAsmIfTyp : 	STRUCT
		Cmd : AcpTrakAsmCmdsTyp;
		Par : AcpTrakAsmParTyp;
		Sts : AcpTrakAsmStsTyp;
	END_STRUCT;
	AcpTrakAsmCmdsTyp : 	STRUCT
		Power : BOOL;
		Run : BOOL;
		Reset : BOOL;
	END_STRUCT;
	AcpTrakAsmParTyp : 	STRUCT
		NumShuttles : USINT;
		Startup : AcpTrakAsmStartupParTyp;
		FirstMove : SystemDestinationsEnum;
	END_STRUCT;
	AcpTrakAsmStartupParTyp : 	STRUCT
		Sector : McSectorType;
		Position : LREAL;
		Gap : LREAL;
	END_STRUCT;
	AcpTrakAsmStsTyp : 	STRUCT
		Powered : BOOL;
		WaitingToStart : BOOL;
		Running : BOOL;
		CurrentShuttleIdx : USINT;
		Error : BOOL;
		ErrorID : UDINT;
	END_STRUCT;
END_TYPE
```

### Global.var - Global variables
```iecst
VAR
	gShuttleMon : McAcpTrakAssemblyMonData;
	gUserData : shUserData;
	gMainIf : MainIfTyp;
	gAsmIf : AcpTrakAsmIfTyp;
	gDestLookups : ARRAY[0..MAX_DESTINATIONS_IDX] OF SystemDestinationsTyp;
END_VAR
```

### Package Logical/Libraries - Global libraries

### Library Logical/Libraries/TrakHelper (IEC)

#### Types.typ - Exported data types
```iecst
(*Shuttle User Data and Other Modifyable Types*)

TYPE
	SystemDestinationsEnum :
		(
		DEST_STARTUP,
		DEST_DECIDE_1 := 5,
		DEST_PROCESS_1 := 10,
		DEST_PROCESS_1A,
		DEST_PROCESS_1B,
		DEST_PROCESS_2 := 20,
		DEST_PROCESS_2A,
		DEST_PROCESS_2B,
		DEST_PROCESS_3 := 30
		);
	shUserData : 	STRUCT
		ColorRGB : ARRAY[0..2]OF REAL;
		ShId : STRING[10];
		Destination : SystemDestinationsEnum;
	END_STRUCT;
	shColors_Typ :
		(
		COLOR_RED,
		COLOR_GREEN,
		COLOR_BLUE,
		COLOR_YELLOW,
		COLOR_WHITE,
		COLOR_ORANGE,
		COLOR_CYAN,
		COLOR_BLACK,
		COLOR_PINK
		);
	SystemDestinationsTyp : 	STRUCT
		Name : STRING[32];
		Sector : McSectorType;
		Position : LREAL;
		ProcPoint : McProcessPointType;
	END_STRUCT;
END_TYPE

(*Process Point Wrapper Type*)

TYPE
	ProcWrapperParTyp : 	STRUCT
		Dest : ProcWrapperDestParTyp;
		DestinationCheck : BOOL;
	END_STRUCT;
	ProcWrapperDestParTyp : 	STRUCT
		Color : shColors_Typ;
		MoveType : ProcWrapperMoveTypes;
		Destination : SystemDestinationsEnum;
		Velocity : REAL;
		Accel : REAL;
		Decel : REAL;
	END_STRUCT;
	ProcWrapperMoveTypes :
		(
		MV_ROUTE_ABSOLUTE,
		MV_ROUTE_VELOCITY,
		MV_ELASTIC_ABSOLUTE,
		MV_ELASTIC_VELOCITY
		);
	ProcWrapperInternalTyp : 	STRUCT
		state : ProcWrapperStatesEnum;
		errorState : ProcWrapperStatesEnum;
		Shuttle : ProcWrapperShInfoTyp;
		Fbs : ProcWrapperIntFbsTyp;
		Test : STRING[80];
	END_STRUCT;
	ProcWrapperShInfoTyp : 	STRUCT
		Axis : McAxisType;
		UserData : shUserData;
	END_STRUCT;
	ProcWrapperIntFbsTyp : 	STRUCT
		RouteVelFb : MC_BR_RoutedMoveVel_AcpTrak;
		RouteAbsFb : MC_BR_RoutedMoveAbs_AcpTrak;
		ElasticVelFb : MC_BR_ElasticMoveVel_AcpTrak;
		ElasticAbsFb : MC_BR_ElasticMoveAbs_AcpTrak;
		ElasticAddFb : MC_BR_ElasticMoveAdd_AcpTrak;
		TrgPtFb : MC_BR_TrgPointEnable_AcpTrak;
		TrgPtGetInfoFb : MC_BR_TrgPointGetInfo_AcpTrak;
		ShCopyDataFb : MC_BR_ShCopyUserData_AcpTrak;
		ShReadInfoFb : MC_BR_ShReadInfo_AcpTrak;
	END_STRUCT;
	ProcWrapperStatesEnum :
		(
		PROC_OFF,
		PROC_INIT,
		PROC_WAIT_SHUTTLE,
		PROC_GET_TRG_INFO,
		PROC_GET_USER_DATA,
		PROC_CHECK,
		PROC_UPDATE_USER_DATA,
		PROC_SEND,
		PROC_ERROR
		);
END_TYPE
```

#### Constants.var - Exported constants
```iecst
VAR CONSTANT
	MAX_SHUTTLE_BUFFER_SIZE : USINT := 5;
	MAX_SHUTTLE_BUFFER_IDX : USINT := MAX_SHUTTLE_BUFFER_SIZE-1;
	MAX_DESTINATIONS : USINT := 255;
	MAX_DESTINATIONS_IDX : USINT := MAX_DESTINATIONS-1;
END_VAR
```

#### TrakHelper.fun - Exported functions and function blocks
```iecst
{REDUND_ERROR} FUNCTION shSetColor : UDINT (*Wrapper to set a RGB color value for a shuttle based upon an enumeration*) (*$GROUP=User,$CAT=User,$GROUPICON=User.png,$CATICON=User.png*)
	VAR_INPUT
		Color : shColors_Typ;
		pRGB : REFERENCE TO ARRAY[0..2] OF REAL;
	END_VAR
END_FUNCTION

{REDUND_ERROR} FUNCTION_BLOCK procWrapper (*TODO: Add your comment here*) (*$GROUP=User,$CAT=User,$GROUPICON=User.png,$CATICON=User.png*)
	VAR_INPUT
		Enable : {REDUND_UNREPLICABLE} BOOL;
		ProcessPt : SystemDestinationsEnum;
		DestLookups : REFERENCE TO ARRAY[0..MAX_DESTINATIONS_IDX] OF SystemDestinationsTyp;
		Pars : REFERENCE TO ProcWrapperParTyp;
	END_VAR
	VAR_OUTPUT
		Active : BOOL;
		Error : BOOL;
		ErrorID : UDINT;
		ShPresent : BOOL;
	END_VAR
	VAR
		int : ProcWrapperInternalTyp;
	END_VAR
END_FUNCTION_BLOCK
```

#### shSetColor.st
```iecst
(* Wrapper to set a RGB color value for a shuttle based upon an enumeration *)
FUNCTION shSetColor
	CASE Color OF
		COLOR_GREEN:
			pRGB[0] := 0.0;
			pRGB[1] := 1.0;
			pRGB[2] := 0.0;
		COLOR_BLUE:
			pRGB[0] := 0.0;
			pRGB[1] := 0.0;
			pRGB[2] := 1.0;
		COLOR_RED:
			pRGB[0] := 1.0;
			pRGB[1] := 0.0;
			pRGB[2] := 0.0;
		COLOR_YELLOW:
			pRGB[0] := 0.8;
			pRGB[1] := 0.8;
			pRGB[2] := 0.0;
		COLOR_WHITE:
			pRGB[0] := 1.0;
			pRGB[1] := 1.0;
			pRGB[2] := 1.0;
		COLOR_ORANGE:
			pRGB[0] := 1.0;
			pRGB[1] := 0.5;
			pRGB[2] := 0;
		COLOR_CYAN:
			pRGB[0] := 0;
			pRGB[1] := 1.0;
			pRGB[2] := 1.0;
		COLOR_BLACK:
			pRGB[0] := 0;
			pRGB[1] := 0;
			pRGB[2] := 0;
		COLOR_PINK:
			pRGB[0] := 1;
			pRGB[1] := 0;
			pRGB[2] := 0.5;
	END_CASE;

END_FUNCTION
```

#### procWrapper.st
```iecst
FUNCTION_BLOCK procWrapper
	//Enable the Trg Point
	//Check for shuttles
	//Read
	IF Enable THEN
		CASE int.state OF
			//************************** Idle/Off/Default State
			PROC_OFF:
				int.Fbs.TrgPtFb.Enable := TRUE;
				int.Fbs.TrgPtFb.ProcessPoint := ADR(DestLookups[ProcessPt].ProcPoint);

				int.state := PROC_INIT;
			//************************** Init State
			PROC_INIT:
				IF int.Fbs.TrgPtFb.Valid THEN
					int.state := PROC_WAIT_SHUTTLE;
				END_IF
				//************************** Waiting For A Shuttle State
			PROC_WAIT_SHUTTLE:
				IF int.Fbs.TrgPtFb.Error THEN
					int.errorState := int.state;
					Error := TRUE;
					ErrorID := int.Fbs.TrgPtFb.ErrorID;
					int.state := PROC_ERROR;
				ELSIF int.Fbs.TrgPtFb.EventCount > 0 THEN
					int.Fbs.TrgPtGetInfoFb.Execute := TRUE;
					int.Fbs.TrgPtGetInfoFb.ProcessPoint := ADR(DestLookups[ProcessPt].ProcPoint);

					int.state := PROC_GET_TRG_INFO;
				END_IF
			//************************** Get Trigger Point Info State
			PROC_GET_TRG_INFO:
				IF int.Fbs.TrgPtGetInfoFb.Error THEN
					int.errorState := int.state;
					Error := TRUE;
					ErrorID := int.Fbs.TrgPtGetInfoFb.ErrorID;
					int.state := PROC_ERROR;
				ELSIF int.Fbs.TrgPtGetInfoFb.Done THEN
					int.Shuttle.Axis := int.Fbs.TrgPtGetInfoFb.TrgPointInfo.Axis;
					int.Fbs.TrgPtGetInfoFb.Execute := FALSE;

					int.Fbs.ShCopyDataFb.Axis := ADR(int.Shuttle.Axis);
					int.Fbs.ShCopyDataFb.DataAddress := ADR(int.Shuttle.UserData);
					int.Fbs.ShCopyDataFb.DataSize := SIZEOF(int.Shuttle.UserData);
					int.Fbs.ShCopyDataFb.Mode := mcACPTRAK_USERDATA_GET;
					int.Fbs.ShCopyDataFb.Execute := TRUE;

					int.Fbs.ShReadInfoFb.Axis := ADR(int.Shuttle.Axis);
					int.Fbs.ShReadInfoFb.Enable := TRUE;

					int.state := PROC_GET_USER_DATA;
				END_IF
			//************************** Getting User Data and Sh Info State
			PROC_GET_USER_DATA:
				IF int.Fbs.ShReadInfoFb.Error OR int.Fbs.ShCopyDataFb.Error THEN
					int.errorState := int.state;
					Error := TRUE;
					int.state := PROC_ERROR;
				ELSIF int.Fbs.ShReadInfoFb.Valid AND int.Fbs.ShCopyDataFb.Done THEN
					int.Fbs.ShCopyDataFb.Execute := FALSE;

					IF int.Fbs.ShReadInfoFb.ShuttleInfo.RouteDestinationInfo.SectorType <> mcACPTRAK_SEC_INTERNAL THEN
						int.state := PROC_CHECK;
					ELSE
						int.Fbs.ShReadInfoFb.Enable := FALSE;
						int.Fbs.TrgPtGetInfoFb.Execute := FALSE;

						brsmemset(ADR(int.Shuttle),0,SIZEOF(int.Shuttle));

						int.state := PROC_WAIT_SHUTTLE;
					END_IF
				END_IF
			//************************** Preforming The Decision State
			PROC_CHECK:
				IF ( Pars.DestinationCheck AND DestLookups[ProcessPt].Sector.controlif = DestLookups[int.Shuttle.UserData.Destination].Sector.controlif)
					OR NOT Pars.DestinationCheck THEN
					ShPresent := TRUE;

					shSetColor(Pars.Dest.Color,ADR(int.Shuttle.UserData.ColorRGB));
					int.Shuttle.UserData.Destination := Pars.Dest.Destination;

					int.Fbs.ShCopyDataFb.Execute := TRUE;
					int.Fbs.ShCopyDataFb.Mode := mcACPTRAK_USERDATA_SET;

					int.state := PROC_UPDATE_USER_DATA;
				ELSE
					int.Fbs.ShReadInfoFb.Enable := FALSE;

					brsmemset(ADR(int.Shuttle),0,SIZEOF(int.Shuttle));

					int.state := PROC_WAIT_SHUTTLE;
				END_IF
			//************************** Updating the User Data State
			PROC_UPDATE_USER_DATA:
				IF int.Fbs.ShCopyDataFb.Error THEN
				ELSIF int.Fbs.ShCopyDataFb.Done THEN
					int.Fbs.ShCopyDataFb.Execute := FALSE;
					int.Test := DestLookups[int.Shuttle.UserData.Destination].Name;
					CASE Pars.Dest.MoveType OF
						MV_ROUTE_ABSOLUTE:
							int.Fbs.RouteAbsFb.Axis := ADR(int.Shuttle.Axis);
							int.Fbs.RouteAbsFb.Sector := ADR(DestLookups[int.Shuttle.UserData.Destination].Sector);
							int.Fbs.RouteAbsFb.Position := DestLookups[int.Shuttle.UserData.Destination].Position;
							int.Fbs.RouteAbsFb.Velocity := Pars.Dest.Velocity;
							int.Fbs.RouteAbsFb.Acceleration := Pars.Dest.Accel;
							int.Fbs.RouteAbsFb.Deceleration := Pars.Dest.Decel;
							int.Fbs.RouteAbsFb.Execute := TRUE;
						MV_ROUTE_VELOCITY:
							int.Fbs.RouteVelFb.Axis := ADR(int.Shuttle.Axis);
							int.Fbs.RouteVelFb.Sector := ADR(DestLookups[int.Shuttle.UserData.Destination].Sector);
							int.Fbs.RouteVelFb.Position := DestLookups[int.Shuttle.UserData.Destination].Position;
							int.Fbs.RouteVelFb.Velocity := Pars.Dest.Velocity;
							int.Fbs.RouteVelFb.RouteVelocity := Pars.Dest.Velocity;
							int.Fbs.RouteVelFb.Acceleration := Pars.Dest.Accel;
							int.Fbs.RouteVelFb.Deceleration := Pars.Dest.Decel;
							int.Fbs.RouteVelFb.Execute := TRUE;
						MV_ELASTIC_ABSOLUTE:
							int.Fbs.ElasticAbsFb.Axis := ADR(int.Shuttle.Axis);
							int.Fbs.ElasticAbsFb.Position := DestLookups[int.Shuttle.UserData.Destination].Position;
							int.Fbs.ElasticAbsFb.Velocity := Pars.Dest.Velocity;
							int.Fbs.ElasticAbsFb.Acceleration := Pars.Dest.Accel;
							int.Fbs.ElasticAbsFb.Deceleration := Pars.Dest.Decel;
							int.Fbs.ElasticAbsFb.Execute := TRUE;
						MV_ELASTIC_VELOCITY:
							int.Fbs.ElasticVelFb.Axis := ADR(int.Shuttle.Axis);
							int.Fbs.ElasticVelFb.Velocity := Pars.Dest.Velocity;
							int.Fbs.ElasticVelFb.Acceleration := Pars.Dest.Accel;
							int.Fbs.ElasticVelFb.Deceleration := Pars.Dest.Decel;
							int.Fbs.ElasticVelFb.Execute := TRUE;
					END_CASE;
					int.state := PROC_SEND;
				END_IF
			//************************** Sending the Shuttle State
			PROC_SEND:
				IF int.Fbs.RouteAbsFb.Error OR
					int.Fbs.RouteVelFb.Error OR
					int.Fbs.ElasticAbsFb.Error OR
					int.Fbs.ElasticVelFb.Error THEN

					int.errorState := int.state;
					Error := TRUE;
					int.state := PROC_ERROR;
				ELSIF NOT int.Fbs.RouteAbsFb.Execute AND
					NOT int.Fbs.RouteVelFb.Execute AND
					NOT int.Fbs.ElasticAbsFb.Execute AND
					NOT int.Fbs.ElasticVelFb.Execute THEN

					ShPresent := FALSE;

					int.Fbs.ShReadInfoFb.Enable := FALSE;
					int.state := PROC_WAIT_SHUTTLE;
				END_IF
			//************************** Error State
			PROC_ERROR:
		END_CASE;
		int.Fbs.ElasticAbsFb();
		int.Fbs.ElasticVelFb();
		int.Fbs.RouteAbsFb();
		int.Fbs.RouteVelFb();
		int.Fbs.ShCopyDataFb();
		int.Fbs.ShReadInfoFb();
		int.Fbs.TrgPtFb();
		int.Fbs.TrgPtGetInfoFb();

		IF int.Fbs.ElasticAbsFb.Active THEN
			int.Fbs.ElasticAbsFb.Execute := FALSE;
		END_IF
		IF int.Fbs.ElasticVelFb.Active THEN
			int.Fbs.ElasticVelFb.Execute := FALSE;
		END_IF
		IF int.Fbs.RouteAbsFb.Active THEN
			int.Fbs.RouteAbsFb.Execute := FALSE;
		END_IF
		IF int.Fbs.RouteVelFb.Active THEN
			int.Fbs.RouteVelFb.Execute := FALSE;
		END_IF

	ELSE

	END_IF
END_FUNCTION_BLOCK
```

### Program Logical/Source/Main (IEC)

#### Cyclic.st - Cyclic code
```iecst
PROGRAM _CYCLIC
	LookupDefine;
	//Main state machine

	//Send cmd to enable Assembly
	//Send cmd to enable stations
	//Send cmd to start process

END_PROGRAM
```

#### Init.st - Init code
```iecst
PROGRAM _INIT
	gMainIf.Par.DefaultAccel := 20.0;
	gMainIf.Par.DefaultDecel := 20.0;
	gMainIf.Par.DefaultVelocity := 2.0;

END_PROGRAM
```

#### LookupDefine.st
```iecst
ACTION LookupDefine:
	//DEST_STARTUP
	gDestLookups[DEST_STARTUP].Name := 'DEST_STARTUP';
	gDestLookups[DEST_STARTUP].Position := 0.0;
	gDestLookups[DEST_STARTUP].Sector := secStartup;
	//gDestLookups[DEST_STARTUP].ProcPoint := ppCellDecision;

	//DEST_DECIDE_1
	gDestLookups[DEST_DECIDE_1].Name := 'DEST_DECIDE_1';
	gDestLookups[DEST_DECIDE_1].Position := 0.0;
	gDestLookups[DEST_DECIDE_1].Sector := secLoadDecision;
	gDestLookups[DEST_DECIDE_1].ProcPoint := ppLoadDecision;

	//DEST_PROCESS_1
	gDestLookups[DEST_PROCESS_1].Name := 'DEST_PROCESS_1';
	gDestLookups[DEST_PROCESS_1].Position := 0.0;
	gDestLookups[DEST_PROCESS_1].Sector := secProcess1;
	gDestLookups[DEST_PROCESS_1].ProcPoint := ppProcess1;

	//DEST_PROCESS_2
	gDestLookups[DEST_PROCESS_2].Name := 'DEST_PROCESS_2';
	gDestLookups[DEST_PROCESS_2].Position := 0.0;
	gDestLookups[DEST_PROCESS_2].Sector := secProcess2;
	gDestLookups[DEST_PROCESS_2].ProcPoint := ppProcess2;
END_ACTION
```

### Program Logical/Source/AssemblyCtrl (IEC)

#### Types.typ
```iecst
TYPE
	AssemblyStatesEnum :
		(
		ASM_IDLE,
		ASM_POWER_ON,
		ASM_CHECK_COUNT,
		ASM_ADD_SHUTTLE,
		ASM_WRITE_DATA,
		ASM_WAIT_START,
		ASM_GET_SHUTTLE,
		ASM_SEND_SHUTTLE,
		ASM_RUNNING,
		ASM_ERROR
		);
	AsmFbsTyp : 	STRUCT
		PowerOnFb : MC_BR_AsmPowerOn_AcpTrak;
		PowerOffFb : MC_BR_AsmPowerOff_AcpTrak;
		SecAddShFb : MC_BR_SecAddShuttle_AcpTrak;
		SecGetShFb : MC_BR_SecGetShuttle_AcpTrak;
		RoutedMoveVelFb : MC_BR_RoutedMoveVel_AcpTrak;
		ShCopyDataFb : MC_BR_ShCopyUserData_AcpTrak;
	END_STRUCT;
END_TYPE
```

#### Variables.var
```iecst
VAR
	state : AssemblyStatesEnum;
	errorState : AssemblyStatesEnum;
	fbs : AsmFbsTyp;
	userData : shUserData;
END_VAR
```

#### Cyclic.st
```iecst
PROGRAM _CYCLIC

	//Idle
	//Power On the assembly
	//Add shuttles
	//Wait Start Command
	//Send all shuttles moving
	//Power Off the assembly
	//Error
	//Reset

	CASE state OF
		//******************************************************************** Idle State
		ASM_IDLE:
			IF gAsmIf.Cmd.Power THEN

				gAsmIf.Sts.CurrentShuttleIdx := 0;
				gAsmIf.Par.Startup.Sector := secStartup;

				fbs.PowerOnFb.Assembly := ADR(gTestAssembly);
				fbs.PowerOnFb.Execute := TRUE;

				state := ASM_POWER_ON;
			END_IF
		//******************************************************************** Power On State
		ASM_POWER_ON:
			IF fbs.PowerOnFb.Error THEN
				errorState := state;
				state := ASM_ERROR;
				gAsmIf.Sts.Error := TRUE;
			ELSIF fbs.PowerOnFb.Done THEN
				fbs.PowerOnFb.Execute := FALSE;
				gAsmIf.Sts.Powered := TRUE;

				state := ASM_CHECK_COUNT;
			END_IF
		//******************************************************************** Adding Shuttles State
		ASM_ADD_SHUTTLE:
			IF fbs.SecAddShFb.Error THEN
				errorState := state;
				state := ASM_ERROR;
				gAsmIf.Sts.Error := TRUE;
			ELSIF fbs.SecAddShFb.Done THEN
				shSetColor(COLOR_GREEN,ADR(userData.ColorRGB));
				brsitoa(USINT_TO_DINT(gAsmIf.Sts.CurrentShuttleIdx),ADR(userData.ShId));
				userData.Destination := DEST_DECIDE_1;

				fbs.ShCopyDataFb.Axis := ADR(fbs.SecAddShFb.Axis);
				fbs.ShCopyDataFb.DataAddress := ADR(userData);
				fbs.ShCopyDataFb.DataSize := SIZEOF(userData);
				fbs.ShCopyDataFb.Mode := mcACPTRAK_USERDATA_SET;
				fbs.ShCopyDataFb.Execute := TRUE;

				state := ASM_WRITE_DATA;
			END_IF
		//******************************************************************** Update Shuttle User Data State
		ASM_WRITE_DATA:
			IF fbs.ShCopyDataFb.Error THEN
				errorState := state;
				state := ASM_ERROR;
				gAsmIf.Sts.Error := TRUE;
			ELSIF fbs.ShCopyDataFb.Done THEN
				fbs.ShCopyDataFb.Execute := FALSE;
				fbs.SecAddShFb.Execute := FALSE;
				gAsmIf.Sts.CurrentShuttleIdx := gAsmIf.Sts.CurrentShuttleIdx + 1;

				state := ASM_CHECK_COUNT;
			END_IF

		//******************************************************************** Check Count State
		ASM_CHECK_COUNT:
			IF gAsmIf.Sts.CurrentShuttleIdx >= gAsmIf.Par.NumShuttles THEN
				gAsmIf.Sts.WaitingToStart := TRUE;

				state := ASM_WAIT_START;
			ELSE
				fbs.SecAddShFb.Sector := ADR(gAsmIf.Par.Startup.Sector);
				fbs.SecAddShFb.Position := gAsmIf.Par.Startup.Position + gAsmIf.Par.Startup.Gap * gAsmIf.Sts.CurrentShuttleIdx;
				fbs.SecAddShFb.Execute := TRUE;

				state := ASM_ADD_SHUTTLE;
			END_IF
		//******************************************************************** Idle State
		ASM_WAIT_START:
			IF gAsmIf.Cmd.Run THEN
				fbs.SecGetShFb.Sector := ADR(gAsmIf.Par.Startup.Sector);
				fbs.SecGetShFb.Mode := mcACPTRAK_SEARCH_BACKWARD;
				fbs.SecGetShFb.Enable := TRUE;

				state := ASM_GET_SHUTTLE;
			END_IF
		//******************************************************************** Idle State
		ASM_GET_SHUTTLE:
			IF fbs.SecGetShFb.Error THEN
				errorState := state;
				state := ASM_ERROR;
				gAsmIf.Sts.Error := TRUE;
			ELSIF fbs.SecGetShFb.Valid THEN
				fbs.SecGetShFb.Next := FALSE;
				fbs.RoutedMoveVelFb.Axis := ADR(fbs.SecGetShFb.Axis);
				fbs.RoutedMoveVelFb.Sector := ADR(gDestLookups[gAsmIf.Par.FirstMove].Sector);
				fbs.RoutedMoveVelFb.Position := gDestLookups[gAsmIf.Par.FirstMove].Position;
				fbs.RoutedMoveVelFb.Velocity := gMainIf.Par.DefaultVelocity;
				fbs.RoutedMoveVelFb.RouteVelocity := gMainIf.Par.DefaultVelocity;
				fbs.RoutedMoveVelFb.Acceleration := gMainIf.Par.DefaultAccel;
				fbs.RoutedMoveVelFb.Deceleration := gMainIf.Par.DefaultDecel;
				fbs.RoutedMoveVelFb.AdvancedParameters.StartDirection := mcDIR_POSITIVE;
				fbs.RoutedMoveVelFb.Execute := TRUE;

				state := ASM_SEND_SHUTTLE;

			END_IF

		//******************************************************************** Idle State
		ASM_SEND_SHUTTLE:
			IF fbs.RoutedMoveVelFb.Error THEN
				errorState := state;
				state := ASM_ERROR;
				gAsmIf.Sts.Error := TRUE;
			ELSIF NOT fbs.RoutedMoveVelFb.Execute THEN
				IF fbs.SecGetShFb.RemainingCount = 0 THEN
					fbs.SecGetShFb.Enable := FALSE;
					fbs.SecGetShFb.Next := FALSE;
					gAsmIf.Sts.Running := TRUE;

					state := ASM_RUNNING;
				ELSE
					fbs.SecGetShFb.Next := TRUE;

					state := ASM_GET_SHUTTLE;
				END_IF
			END_IF
		//******************************************************************** Idle State
		ASM_RUNNING:
		//******************************************************************** Idle State
		ASM_ERROR:

	END_CASE;

	fbs.PowerOnFb();
	fbs.RoutedMoveVelFb();
	fbs.SecAddShFb();
	fbs.SecGetShFb();
	fbs.ShCopyDataFb();

	IF fbs.RoutedMoveVelFb.Active THEN
		fbs.RoutedMoveVelFb.Execute := FALSE;
	END_IF
END_PROGRAM
```

#### Init.st
```iecst
PROGRAM _INIT
	gAsmIf.Par.NumShuttles := 20;
	gAsmIf.Par.Startup.Position := 0;
	gAsmIf.Par.Startup.Gap := 0.06;
	gAsmIf.Par.FirstMove := DEST_DECIDE_1;

END_PROGRAM
```

### Library Logical/Source/Stations/ProcLogic (IEC) - Station Logic Library

#### Types.typ - Exported data types
```iecst
TYPE
	DeciderStationIntTyp : 	STRUCT
		state : DeciderStationStateEnum;
		errorState : DeciderStationStateEnum;
		currentIdx : USINT;
		Fbs : DeciderStationFbTyp;
	END_STRUCT;
	DeciderStationStateEnum :
		(
		DECIDER_OFF,
		DECIDER_INIT,
		DECIDER_WAIT,
		DECIDER_PROCESS_SHUTTLE,
		DECIDER_ERROR
		);
	DeciderStationFbTyp : 	STRUCT
		procWrapperFb : procWrapper;
	END_STRUCT;
END_TYPE
```

#### Constants.var - Exported constants
```iecst
VAR CONSTANT
	MAX_DECIDERS_IDX : USINT := MAX_DECIDERS_COUNT-1;
	MAX_DECIDERS_COUNT : USINT := 5;
END_VAR
```

#### ProcLogic.fun - Exported functions and function blocks
```iecst
{REDUND_ERROR} FUNCTION_BLOCK DeciderStationFb (*TODO: Add your comment here*) (*$GROUP=User,$CAT=User,$GROUPICON=User.png,$CATICON=User.png*)
	VAR_INPUT
		Enable : {REDUND_UNREPLICABLE} BOOL;
		ProcPt : SystemDestinationsEnum;
		DestLookup : REFERENCE TO ARRAY[0..MAX_DESTINATIONS_IDX] OF SystemDestinationsTyp;
		DestList : {REDUND_UNREPLICABLE} ARRAY[0..MAX_DECIDERS_IDX] OF SystemDestinationsEnum;
		NumberOfDestinations : USINT;
		StationPars : ProcWrapperParTyp;
	END_VAR
	VAR_OUTPUT
		Active : BOOL;
		NextDest : SystemDestinationsEnum;
		Error : BOOL;
		ErrorID : BOOL;
	END_VAR
	VAR
		int : DeciderStationIntTyp;
	END_VAR
END_FUNCTION_BLOCK
```

#### DeciderStationFb.st
```iecst
(* TODO: Add your comment here *)
FUNCTION_BLOCK DeciderStationFb
	CASE int.state OF
		//*************************** Off/Idle State
		DECIDER_OFF:
			IF Enable THEN
				int.currentIdx := 0;
				StationPars.Dest.Destination := DestList[int.currentIdx];

				int.Fbs.procWrapperFb.Enable := TRUE;
				int.Fbs.procWrapperFb.Pars := ADR(StationPars);
				int.Fbs.procWrapperFb.DestLookups := ADR(DestLookup);
				int.Fbs.procWrapperFb.ProcessPt := ProcPt;
				int.state := DECIDER_INIT;
			END_IF
		//*************************** Init State
		DECIDER_INIT:
			int.state := DECIDER_WAIT;

		//*************************** Waiting for a shuttle State
		DECIDER_WAIT:
			IF int.Fbs.procWrapperFb.ShPresent THEN
				int.state := DECIDER_PROCESS_SHUTTLE;
			END_IF
		//*************************** Processing the Shuttle State
		DECIDER_PROCESS_SHUTTLE:
			IF NOT int.Fbs.procWrapperFb.ShPresent THEN
				int.currentIdx := int.currentIdx + 1;
				IF int.currentIdx > MAX_DECIDERS_IDX OR int.currentIdx + 1 > NumberOfDestinations THEN
					int.currentIdx := 0;
				END_IF

				StationPars.Dest.Destination := DestList[int.currentIdx];
				int.state := DECIDER_WAIT;
			END_IF
	END_CASE;

	NextDest := DestList[int.currentIdx];

	int.Fbs.procWrapperFb();

END_FUNCTION_BLOCK
```

### Program Logical/Source/Stations/Deciders (IEC)

#### Variables.var
```iecst
VAR
	loopDeciderFb : DeciderStationFb;
	proc2Fb : DeciderStationFb;
	proc1Fb : DeciderStationFb;
END_VAR
```

#### Cyclic.st
```iecst
PROGRAM _CYCLIC

	loopDeciderFb.Enable := gAsmIf.Cmd.Run;
	proc1Fb.Enable := gAsmIf.Cmd.Run;
	proc2Fb.Enable := gAsmIf.Cmd.Run;

	loopDeciderFb();
	proc1Fb();
	proc2Fb();
END_PROGRAM
```

#### Init.st
```iecst
PROGRAM _INIT
	loopDeciderFb.DestList[0] := DEST_PROCESS_1;
	loopDeciderFb.DestList[1] := DEST_PROCESS_2;
	loopDeciderFb.NumberOfDestinations := 2;
	loopDeciderFb.ProcPt := DEST_DECIDE_1;
	loopDeciderFb.DestLookup := ADR(gDestLookups);

	loopDeciderFb.StationPars.Dest.Accel := 20.0;
	loopDeciderFb.StationPars.Dest.Decel := 20.0;
	loopDeciderFb.StationPars.Dest.Velocity := 1.0;
	loopDeciderFb.StationPars.Dest.MoveType := MV_ROUTE_VELOCITY;
	loopDeciderFb.StationPars.Dest.Color := COLOR_CYAN;

	proc1Fb.DestList[0] := DEST_DECIDE_1;
	proc1Fb.NumberOfDestinations := 1;
	proc1Fb.ProcPt := DEST_PROCESS_1;
	proc1Fb.DestLookup := ADR(gDestLookups);

	proc1Fb.StationPars.Dest.Accel := 20.0;
	proc1Fb.StationPars.Dest.Decel := 20.0;
	proc1Fb.StationPars.Dest.Velocity := 1.5;
	proc1Fb.StationPars.Dest.MoveType := MV_ROUTE_VELOCITY;
	proc1Fb.StationPars.Dest.Color := COLOR_YELLOW;

	proc2Fb.DestList[0] := DEST_DECIDE_1;
	proc2Fb.NumberOfDestinations := 1;
	proc2Fb.ProcPt := DEST_PROCESS_2;
	proc2Fb.DestLookup := ADR(gDestLookups);

	proc2Fb.StationPars.Dest.Accel := 20.0;
	proc2Fb.StationPars.Dest.Decel := 20.0;
	proc2Fb.StationPars.Dest.Velocity := 1.5;
	proc2Fb.StationPars.Dest.MoveType := MV_ROUTE_VELOCITY;
	proc2Fb.StationPars.Dest.Color := COLOR_RED;

END_PROGRAM
```

### Program Logical/Source/Vis/Vis (IEC)

#### Types.typ
```iecst
(*Visualization to Scene viewer types*)

TYPE
	Stations : 	STRUCT
		Load : Station_Typ;
	END_STRUCT;
	Vis_typ : 	STRUCT
		Trak : McAcpTrakAssemblyVisData;
		A1HumanStation1 : BOOL;
		A1HumanStation2 : BOOL;
		A2HumanStation1 : BOOL;
		A2HumanStation2 : BOOL;
	END_STRUCT;
	Scn_Color_typ : 	STRUCT  (*RGB Strucuture for the scene*)
		Red : REAL;
		Green : REAL;
		Blue : REAL;
	END_STRUCT;
	Station_Typ : 	STRUCT
		Active : BOOL;
		TimeRemaining : STRING[31];
	END_STRUCT;
END_TYPE
```

#### Variables.var
```iecst
VAR
	Vis : Vis_typ;
	SizeofVis : UDINT;
	NumVisShuttle : USINT;
	i : USINT;
	pUserData : REFERENCE TO shUserData;
	index : UINT;
	numShuttles : USINT;
	userDataSize : UDINT;
END_VAR
```

#### Main.st
```iecst
PROGRAM _INIT

    // size of Vis.Trak structure - this value has to be entered in B&R scene viewer (PVI -> Options -> Size)
	SizeofVis := SIZEOF(Vis.Trak);

	userDataSize := SIZEOF(gUserData);

	// max number of displayed shuttles
	NumVisShuttle := SIZEOF(Vis.Trak.Shuttle) / SIZEOF(Vis.Trak.Shuttle[0]);

END_PROGRAM

PROGRAM _CYCLIC

	//Problem with my approach is that we can't easily power cycle due to only wanting to be on the first 10 shuttles, need to fix this by using some modulus or something?

	FOR i:=0 TO (NumVisShuttle-1) DO

		IF gShuttleMon.Shuttle[i].Available THEN
			// format selected monitor data to fit B&R scene viewer
			//This is done to normalize the indecies, make sure we the scene viewer shuttles 1-20 always line up with shuttle index 1-20
			//			index := gShuttleMon.Shuttle[i].Index-1;
			//			index := index MOD numShuttles;
			CASE index OF
				0..19:
					Vis.Trak.Shuttle[i].Available    	:= 1;
					Vis.Trak.Shuttle[i].PositionX    	:= LREAL_TO_REAL(gShuttleMon.Shuttle[i].Position.X);
					Vis.Trak.Shuttle[i].PositionY    	:= LREAL_TO_REAL(gShuttleMon.Shuttle[i].Position.Y);
					Vis.Trak.Shuttle[i].RotationZ    	:= LREAL_TO_REAL(gShuttleMon.Shuttle[i].Orientation.Angle1);
					Vis.Trak.Shuttle[i].ExtentToFront    := LREAL_TO_REAL(gShuttleMon.Shuttle[i].ExtentToFront);
					Vis.Trak.Shuttle[i].ExtentToBack     := LREAL_TO_REAL(gShuttleMon.Shuttle[i].ExtentToBack);
					Vis.Trak.Shuttle[i].Width    		:= LREAL_TO_REAL(gShuttleMon.Shuttle[i].Width);
				20..21:
					Vis.Trak.Shuttle[i].Available    	:= 1;
					Vis.Trak.Shuttle[i].PositionX    	:= LREAL_TO_REAL(gShuttleMon.Shuttle[i].Position.Z);
					Vis.Trak.Shuttle[i].PositionY    	:= LREAL_TO_REAL(gShuttleMon.Shuttle[i].Position.Y);
					Vis.Trak.Shuttle[i].RotationZ    	:= LREAL_TO_REAL(gShuttleMon.Shuttle[i].Orientation.Angle1);
					Vis.Trak.Shuttle[i].ExtentToFront    := LREAL_TO_REAL(gShuttleMon.Shuttle[i].ExtentToFront);
					Vis.Trak.Shuttle[i].ExtentToBack     := LREAL_TO_REAL(gShuttleMon.Shuttle[i].ExtentToBack);
					Vis.Trak.Shuttle[i].Width    		:= LREAL_TO_REAL(gShuttleMon.Shuttle[i].Width);
			END_CASE;

			brsitoa(gShuttleMon.Shuttle[i].Index, ADR(Vis.Trak.Shuttle[i].Text));

			// example: set shuttle colour via user data
//			IF gShuttleMon.Shuttle[i].UserData <> 0 THEN
//				pUserData ACCESS gShuttleMon.Shuttle[i].UserData;    // access to user data of this shuttle
//				IF pUserData.ColorEnum = COLOR_GREEN THEN    // product 1 -> display shuttle in green color
//					pUserData.ColorRGB[0]    := 0.0;
//					pUserData.ColorRGB[1]    := 1.0;
//					pUserData.ColorRGB[2]    := 0.0;
//				ELSIF pUserData.ColorEnum = COLOR_BLUE THEN    // product 2 -> display shuttle in blue color
//					pUserData.ColorRGB[0]    := 0.0;
//					pUserData.ColorRGB[1]    := 0.0;
//					pUserData.ColorRGB[2]    := 1.0;
//				ELSIF pUserData.ColorEnum = COLOR_RED THEN    // product 3 -> display shuttle in red color
//					pUserData.ColorRGB[0]    := 1.0;
//					pUserData.ColorRGB[1]    := 0.0;
//					pUserData.ColorRGB[2]    := 0.0;
//				ELSIF pUserData.ColorEnum = COLOR_YELLOW THEN
//					pUserData.ColorRGB[0]    := 0.8;
//					pUserData.ColorRGB[1]    := 0.8;
//					pUserData.ColorRGB[2]    := 0.0;
//				ELSIF pUserData.ColorEnum = COLOR_WHITE THEN
//					pUserData.ColorRGB[0]    := 1.0;
//					pUserData.ColorRGB[1]    := 1.0;
//					pUserData.ColorRGB[2]    := 1.0;
//				ELSIF pUserData.ColorEnum = COLOR_ORANGE THEN
//					pUserData.ColorRGB[0]    := 1.0;
//					pUserData.ColorRGB[1]    := 0.5;
//					pUserData.ColorRGB[2]    := 0;
//				ELSIF pUserData.ColorEnum = COLOR_CYAN THEN
//					pUserData.ColorRGB[0]    := 0;
//					pUserData.ColorRGB[1]    := 1.0;
//					pUserData.ColorRGB[2]    := 1.0;
//				ELSIF pUserData.ColorEnum = COLOR_BLACK THEN
//					pUserData.ColorRGB[0]    := 0;
//					pUserData.ColorRGB[1]    := 0;
//					pUserData.ColorRGB[2]    := 0;
//				ELSIF pUserData.ColorEnum = COLOR_PINK THEN
//					pUserData.ColorRGB[0]    := 1;
//					pUserData.ColorRGB[1]    := 0;
//					pUserData.ColorRGB[2]    := 0.5;
//				END_IF
//			END_IF

		ELSE
			brsmemset(ADR(Vis.Trak.Shuttle[i]), 0, SIZEOF(Vis.Trak.Shuttle[0]));
		END_IF

	END_FOR

END_PROGRAM
```

### Program Logical/Source/Diagnostic/TrakDiag

#### Variables.var
```iecst
VAR
	MC_BR_ShCopyUserData_AcpTrak_0 : MC_BR_ShCopyUserData_AcpTrak;
	ShuttleUserData : shUserData;
	ErrorCodeIDInfo : ARRAY[0..NUM_SEG] OF McAcpTrakSegProcessParIDType;
	SegWarningCmdIDInfo : McAcpTrakSegProcessParIDType;
	SegErrorCheck : ARRAY[0..NUM_SEG] OF SegErrorCheckType;
	CpuSim : BOOL;
END_VAR
(*For testing only*)
VAR
	MC_BR_SegCommandError_AcpTrak_0 : MC_BR_SegCommandError_AcpTrak;
END_VAR
(*Declarations for TrakMap*)
VAR
	paperCore : TrkPaperCore;
	paperOptions : TrkPaperCoreOptionsType;
	TrakDiag : TrkDiagStatusType;
	DiagFbs : DiagFbsType;
	SegIndex : USINT;
END_VAR
```

#### Cyclic.st
```iecst
PROGRAM _CYCLIC

	MC_BR_SegCommandError_AcpTrak_0(Segment := ADR(TrakDiag.Seg.SegList[0].McType));

	IF MC_BR_SegCommandError_AcpTrak_0.Done THEN
		MC_BR_SegCommandError_AcpTrak_0.Execute := FALSE;
	END_IF

	(***********************************ASSEMBLY INFORMATION******************************	)
	(*Read Assebly Status*)

	DiagFbs.Asm.ReadStatus.Enable	:= TRUE;
	DiagFbs.Asm.ReadStatus();

	IF DiagFbs.Asm.ReadStatus.Valid THEN
		TrakDiag.Asm.AssemblyDisabled 	:= DiagFbs.Asm.ReadStatus.AssemblyDisabled;
		TrakDiag.Asm.AssemblyErrorStop := DiagFbs.Asm.ReadStatus.AssemblyErrorStop;
		TrakDiag.Asm.AssemblyReady		:= DiagFbs.Asm.ReadStatus.AssemblyReady;
		TrakDiag.Asm.AssemblyHoming	:= DiagFbs.Asm.ReadStatus.AssemblyHoming;
		TrakDiag.Asm.AssemblyStopping	:= DiagFbs.Asm.ReadStatus.AssemblyStopping;
	END_IF

	(*Read Assembly Info *)

	DiagFbs.Asm.ReadInfo.Enable		:= TRUE;
	DiagFbs.Asm.ReadInfo();

	IF DiagFbs.Asm.ReadInfo.Valid THEN
		TrakDiag.Asm.CommunicationReady 	:= DiagFbs.Asm.ReadInfo.AssemblyInfo.CommunicationReady;
		TrakDiag.Asm.PowerOn				:= DiagFbs.Asm.ReadInfo.AssemblyInfo.PowerOn;
		TrakDiag.Asm.ReadyForPowerOn		:= DiagFbs.Asm.ReadInfo.AssemblyInfo.ReadyForPowerOn;
		TrakDiag.Asm.ShuttlesCount 			:= DiagFbs.Asm.ReadInfo.AssemblyInfo.ShuttlesCount;
		TrakDiag.Asm.ShuttleInErrorStopCount := DiagFbs.Asm.ReadInfo.AssemblyInfo.ShuttlesInErrorStopCount;
		TrakDiag.Asm.StartupCount			:= DiagFbs.Asm.ReadInfo.AssemblyInfo.StartupCount;
	END_IF

	(****************************** SEGMENT ERROR INFORMATION *****************************************)

	FOR SegIndex := 0 TO NUM_SEG DO

		IF TrakDiag.Seg.SegList[SegIndex].McType.controlif <> 0 THEN //If the array contains a segment reference

			DiagFbs.Seg.ReadInfo[SegIndex].Segment 	:= ADR(TrakDiag.Seg.SegList[SegIndex].McType);
			DiagFbs.Seg.ReadInfo[SegIndex].Enable	:= TRUE;
			DiagFbs.Seg.ReadInfo[SegIndex]();

			IF DiagFbs.Seg.ReadInfo[SegIndex].Valid THEN
				//Capture Segment Info
				TrakDiag.Seg.SegList[SegIndex].Status.CommunicationReady 	:= DiagFbs.Seg.ReadInfo[SegIndex].SegmentInfo.CommunicationReady;
				TrakDiag.Seg.SegList[SegIndex].Status.ReadyForPowerOn		:= DiagFbs.Seg.ReadInfo[SegIndex].SegmentInfo.ReadyForPowerOn;
				TrakDiag.Seg.SegList[SegIndex].Status.PowerOn				:= DiagFbs.Seg.ReadInfo[SegIndex].SegmentInfo.PowerOn;
				TrakDiag.Seg.SegList[SegIndex].Status.StartupCount			:= DiagFbs.Seg.ReadInfo[SegIndex].SegmentInfo.StartupCount;
				TrakDiag.Seg.SegList[SegIndex].Status.CommunicationState	:= DiagFbs.Seg.ReadInfo[SegIndex].SegmentInfo.CommunicationState;

			END_IF

			DiagFbs.Seg.ReadStatus[SegIndex].Segment := ADR(TrakDiag.Seg.SegList[SegIndex].McType);
			DiagFbs.Seg.ReadStatus[SegIndex].Enable	:= TRUE;
			DiagFbs.Seg.ReadStatus[SegIndex]();

			IF DiagFbs.Seg.ReadStatus[SegIndex].Valid THEN

				//Check for change of state to ErrorStop to command reading error data, IF communication is ready
				IF ((TrakDiag.Seg.SegList[SegIndex].Status.SegmentErrorStop = FALSE AND DiagFbs.Seg.ReadStatus[SegIndex].SegmentErrorStop = TRUE))
					AND (TrakDiag.Seg.SegList[SegIndex].Status.CommunicationReady = TRUE) THEN

					SegErrorCheck[SegIndex].CmdCheckErrorCode := TRUE;

					//Check for change of state from ErrorStop to reset error number in diag structure
				ELSIF ((TrakDiag.Seg.SegList[SegIndex].Status.SegmentErrorStop = TRUE) AND (DiagFbs.Seg.ReadStatus[SegIndex].SegmentErrorStop = FALSE))
					AND (TrakDiag.Seg.SegList[SegIndex].Status.CommunicationReady = TRUE) THEN

					TrakDiag.Seg.SegList[SegIndex].Status.ErrorCode := 0;

				END_IF
				//Capture Segment Status

				TrakDiag.Seg.SegList[SegIndex].Status.SegmentDisabled	:= DiagFbs.Seg.ReadStatus[SegIndex].SegmentDisabled;
				TrakDiag.Seg.SegList[SegIndex].Status.SegmentErrorStop	:= DiagFbs.Seg.ReadStatus[SegIndex].SegmentErrorStop;
				TrakDiag.Seg.SegList[SegIndex].Status.SegmentReady		:= DiagFbs.Seg.ReadStatus[SegIndex].SegmentReady;
				TrakDiag.Seg.SegList[SegIndex].Status.SegmentStopping	:= DiagFbs.Seg.ReadStatus[SegIndex].SegmentStopping;
			END_IF
		END_IF
	END_FOR

	CpuSim := DiagCpuIsSimulated() OR DiagCpuIsARsim();

	IF CpuSim = FALSE THEN
		actCheckErrorCode;
	END_IF

	(***********************************TRAKMAP******************************)

	//Fetch ShuttleUserData Example

	(* This will likely change to match your project! This is just an example of how to use the
		the click to get a shuttle's user data. The inputs to the ShCopyUserData will reflect your own project
	*)
	IF EDGEPOS(paperCore.ClickData.Shuttle.Valid) THEN
		MC_BR_ShCopyUserData_AcpTrak_0.Axis         := ADR(paperCore.ClickData.Shuttle.Data.Axis);
		MC_BR_ShCopyUserData_AcpTrak_0.Execute      := TRUE;
		MC_BR_ShCopyUserData_AcpTrak_0.DataAddress  := ADR(ShuttleUserData);
		MC_BR_ShCopyUserData_AcpTrak_0.DataSize     := SIZEOF(ShuttleUserData);
		MC_BR_ShCopyUserData_AcpTrak_0.Mode         := mcACPTRAK_USERDATA_GET;
	END_IF

	paperCore();

	MC_BR_ShCopyUserData_AcpTrak_0();
	MC_BR_ShCopyUserData_AcpTrak_0.Execute := FALSE;

END_PROGRAM
```

#### Init.st
```iecst
PROGRAM _INIT

	SegDefinition;

	paperCore.SegmentCount := TrakDiag.Seg.SegCount;
	paperCore.Segments := ADR(TrakDiag.Seg.SegList);
	paperCore.Options := ADR(paperOptions);
	paperCore.Enable := TRUE;
	paperCore.TrakStatus := ADR(TrakDiag);

	(****** Change variables to match your project **********)

	paperCore.Assembly := ADR(gTestAssembly);
	paperCore.ShuttleMon := ADR(gShuttleMon);

	(****************************** Change options here ***********************)

	paperOptions.Color.Offset := 0;
	paperOptions.Segment.Enabled := TRUE;
	paperOptions.Shuttle.Enabled := TRUE;
	paperOptions.Color.Enabled := TRUE;
END_PROGRAM
```

#### SegDefinition.st
```iecst
//This file was automatically generated using the TrakMapImporter program. Verify that the segment names and assembly name match your project values correctly
ACTION SegDefinition:
	TrakDiag.Seg.SegList[0].Name  := 'gCenterLoop_0';		TrakDiag.Seg.SegList[0].McType := gCenterLoop_0;
	TrakDiag.Seg.SegList[1].Name  := 'gCenterLoop_1';		TrakDiag.Seg.SegList[1].McType := gCenterLoop_1;
	TrakDiag.Seg.SegList[2].Name  := 'gCenterLoop_2';		TrakDiag.Seg.SegList[2].McType := gCenterLoop_2;
	TrakDiag.Seg.SegList[3].Name  := 'gCenterLoop_3';		TrakDiag.Seg.SegList[3].McType := gCenterLoop_3;
	TrakDiag.Seg.SegList[4].Name  := 'gCenterLoop_4';		TrakDiag.Seg.SegList[4].McType := gCenterLoop_4;
	TrakDiag.Seg.SegList[5].Name  := 'gCenterLoop_5';		TrakDiag.Seg.SegList[5].McType := gCenterLoop_5;
	TrakDiag.Seg.SegList[6].Name  := 'gCenterLoop_6';		TrakDiag.Seg.SegList[6].McType := gCenterLoop_6;
	TrakDiag.Seg.SegList[7].Name  := 'gCenterLoop_7';		TrakDiag.Seg.SegList[7].McType := gCenterLoop_7;
	TrakDiag.Seg.SegList[8].Name  := 'gCenterLoop_8';		TrakDiag.Seg.SegList[8].McType := gCenterLoop_8;
	TrakDiag.Seg.SegList[9].Name  := 'gCenterLoop_9';		TrakDiag.Seg.SegList[9].McType := gCenterLoop_9;
	TrakDiag.Seg.SegList[10].Name  := 'gCenterLoop_10';		TrakDiag.Seg.SegList[10].McType := gCenterLoop_10;
	TrakDiag.Seg.SegList[11].Name  := 'gCenterLoop_11';		TrakDiag.Seg.SegList[11].McType := gCenterLoop_11;
	TrakDiag.Seg.SegList[12].Name  := 'gCenterLoop_12';		TrakDiag.Seg.SegList[12].McType := gCenterLoop_12;
	TrakDiag.Seg.SegList[13].Name  := 'gCenterLoop_13';		TrakDiag.Seg.SegList[13].McType := gCenterLoop_13;
	TrakDiag.Seg.SegList[14].Name  := 'gCenterLoop_14';		TrakDiag.Seg.SegList[14].McType := gCenterLoop_14;
	TrakDiag.Seg.SegList[15].Name  := 'gCenterLoop_15';		TrakDiag.Seg.SegList[15].McType := gCenterLoop_15;
	TrakDiag.Seg.SegList[16].Name  := 'gCenterLoop_16';		TrakDiag.Seg.SegList[16].McType := gCenterLoop_16;
	TrakDiag.Seg.SegList[17].Name  := 'gCenterLoop_17';		TrakDiag.Seg.SegList[17].McType := gCenterLoop_17;
	TrakDiag.Seg.SegList[18].Name  := 'gCenterLoop_18';		TrakDiag.Seg.SegList[18].McType := gCenterLoop_18;
	TrakDiag.Seg.SegList[19].Name  := 'gCenterLoop_19';		TrakDiag.Seg.SegList[19].McType := gCenterLoop_19;
	TrakDiag.Seg.SegList[20].Name  := 'gCenterLoop_20';		TrakDiag.Seg.SegList[20].McType := gCenterLoop_20;
	TrakDiag.Seg.SegList[21].Name  := 'gCenterLoop_21';		TrakDiag.Seg.SegList[21].McType := gCenterLoop_21;
	TrakDiag.Seg.SegList[22].Name  := 'gCenterLoop_22';		TrakDiag.Seg.SegList[22].McType := gCenterLoop_22;
	TrakDiag.Seg.SegList[23].Name  := 'gCenterLoop_23';		TrakDiag.Seg.SegList[23].McType := gCenterLoop_23;
	TrakDiag.Seg.SegList[24].Name  := 'gCenterLoop_24';		TrakDiag.Seg.SegList[24].McType := gCenterLoop_24;
	TrakDiag.Seg.SegList[25].Name  := 'gCenterLoop_25';		TrakDiag.Seg.SegList[25].McType := gCenterLoop_25;
	TrakDiag.Seg.SegList[26].Name  := 'gCenterLoop_26';		TrakDiag.Seg.SegList[26].McType := gCenterLoop_26;
	TrakDiag.Seg.SegList[27].Name  := 'gCenterLoop_27';		TrakDiag.Seg.SegList[27].McType := gCenterLoop_27;
	TrakDiag.Seg.SegList[28].Name  := 'gCenterLoop_28';		TrakDiag.Seg.SegList[28].McType := gCenterLoop_28;
	TrakDiag.Seg.SegList[29].Name  := 'gCenterLoop_29';		TrakDiag.Seg.SegList[29].McType := gCenterLoop_29;
	TrakDiag.Seg.SegList[30].Name  := 'gCenterLoop_30';		TrakDiag.Seg.SegList[30].McType := gCenterLoop_30;
	TrakDiag.Seg.SegList[31].Name  := 'gCenterLoop_31';		TrakDiag.Seg.SegList[31].McType := gCenterLoop_31;
	TrakDiag.Seg.SegList[32].Name  := 'gCenterLoop_32';		TrakDiag.Seg.SegList[32].McType := gCenterLoop_32;
	TrakDiag.Seg.SegList[33].Name  := 'gCenterLoop_33';		TrakDiag.Seg.SegList[33].McType := gCenterLoop_33;
	TrakDiag.Seg.SegList[34].Name  := 'gCell1_Enter_0';		TrakDiag.Seg.SegList[34].McType := gCell1_Enter_0;
	TrakDiag.Seg.SegList[35].Name  := 'gCell1_Enter_1';		TrakDiag.Seg.SegList[35].McType := gCell1_Enter_1;
	TrakDiag.Seg.SegList[36].Name  := 'gCell1_Load_0';		TrakDiag.Seg.SegList[36].McType := gCell1_Load_0;
	TrakDiag.Seg.SegList[37].Name  := 'gCell1_Load_1';		TrakDiag.Seg.SegList[37].McType := gCell1_Load_1;
	TrakDiag.Seg.SegList[38].Name  := 'gCell1_Load_2';		TrakDiag.Seg.SegList[38].McType := gCell1_Load_2;
	TrakDiag.Seg.SegList[39].Name  := 'gCell1_Load_3';		TrakDiag.Seg.SegList[39].McType := gCell1_Load_3;
	TrakDiag.Seg.SegList[40].Name  := 'gCell1_Load_4';		TrakDiag.Seg.SegList[40].McType := gCell1_Load_4;
	TrakDiag.Seg.SegList[41].Name  := 'gCell1_Load_5';		TrakDiag.Seg.SegList[41].McType := gCell1_Load_5;
	TrakDiag.Seg.SegList[42].Name  := 'gCell1_Load_6';		TrakDiag.Seg.SegList[42].McType := gCell1_Load_6;
	TrakDiag.Seg.SegList[43].Name  := 'gCell1_Load_7';		TrakDiag.Seg.SegList[43].McType := gCell1_Load_7;
	TrakDiag.Seg.SegList[44].Name  := 'gCell1_Load_8';		TrakDiag.Seg.SegList[44].McType := gCell1_Load_8;
	TrakDiag.Seg.SegList[45].Name  := 'gCell1_Load_9';		TrakDiag.Seg.SegList[45].McType := gCell1_Load_9;
	TrakDiag.Seg.SegList[46].Name  := 'gCell1_Load_10';		TrakDiag.Seg.SegList[46].McType := gCell1_Load_10;
	TrakDiag.Seg.SegList[47].Name  := 'gCell1_Exit_0';		TrakDiag.Seg.SegList[47].McType := gCell1_Exit_0;
	TrakDiag.Seg.SegList[48].Name  := 'gCell1_Exit_1';		TrakDiag.Seg.SegList[48].McType := gCell1_Exit_1;
	TrakDiag.Seg.SegList[49].Name  := 'gCell1_Exit_2';		TrakDiag.Seg.SegList[49].McType := gCell1_Exit_2;
	TrakDiag.Seg.SegList[50].Name  := 'gCell1_Exit_3';		TrakDiag.Seg.SegList[50].McType := gCell1_Exit_3;
	TrakDiag.Seg.SegList[51].Name  := 'gCell2_Enter_0';		TrakDiag.Seg.SegList[51].McType := gCell2_Enter_0;
	TrakDiag.Seg.SegList[52].Name  := 'gCell2_Enter_1';		TrakDiag.Seg.SegList[52].McType := gCell2_Enter_1;
	TrakDiag.Seg.SegList[53].Name  := 'gCell2_Load_0';		TrakDiag.Seg.SegList[53].McType := gCell2_Load_0;
	TrakDiag.Seg.SegList[54].Name  := 'gCell2_Load_1';		TrakDiag.Seg.SegList[54].McType := gCell2_Load_1;
	TrakDiag.Seg.SegList[55].Name  := 'gCell2_Load_2';		TrakDiag.Seg.SegList[55].McType := gCell2_Load_2;
	TrakDiag.Seg.SegList[56].Name  := 'gCell2_Load_3';		TrakDiag.Seg.SegList[56].McType := gCell2_Load_3;
	TrakDiag.Seg.SegList[57].Name  := 'gCell2_Load_4';		TrakDiag.Seg.SegList[57].McType := gCell2_Load_4;
	TrakDiag.Seg.SegList[58].Name  := 'gCell2_Load_5';		TrakDiag.Seg.SegList[58].McType := gCell2_Load_5;
	TrakDiag.Seg.SegList[59].Name  := 'gCell2_Load_6';		TrakDiag.Seg.SegList[59].McType := gCell2_Load_6;
	TrakDiag.Seg.SegList[60].Name  := 'gCell2_Load_7';		TrakDiag.Seg.SegList[60].McType := gCell2_Load_7;
	TrakDiag.Seg.SegList[61].Name  := 'gCell2_Load_8';		TrakDiag.Seg.SegList[61].McType := gCell2_Load_8;
	TrakDiag.Seg.SegList[62].Name  := 'gCell2_Load_9';		TrakDiag.Seg.SegList[62].McType := gCell2_Load_9;
	TrakDiag.Seg.SegList[63].Name  := 'gCell2_Load_10';		TrakDiag.Seg.SegList[63].McType := gCell2_Load_10;
	TrakDiag.Seg.SegList[64].Name  := 'gCell2_Exit_0';		TrakDiag.Seg.SegList[64].McType := gCell2_Exit_0;
	TrakDiag.Seg.SegList[65].Name  := 'gCell2_Exit_1';		TrakDiag.Seg.SegList[65].McType := gCell2_Exit_1;
	TrakDiag.Seg.SegList[66].Name  := 'gCell2_Exit_2';		TrakDiag.Seg.SegList[66].McType := gCell2_Exit_2;
	TrakDiag.Seg.SegList[67].Name  := 'gCell2_Exit_3';		TrakDiag.Seg.SegList[67].McType := gCell2_Exit_3;

	TrakDiag.Seg.SegCount := 68;

	TrakDiag.Seg.SegListAdr := ADR(TrakDiag.Seg.SegList);

	DiagFbs.Asm.ReadInfo.Assembly := ADR(gTestAssembly);
	DiagFbs.Asm.ReadStatus.Assembly := ADR(gTestAssembly);

	paperCore.ViewBoxCfg.MinX := -8.65558;
	paperCore.ViewBoxCfg.MinY := -0.745;
	paperCore.ViewBoxCfg.Width := 9.39115;
	paperCore.ViewBoxCfg.Height := 0.86;
END_ACTION
```

### Destinations.typ - not listed in the package file held
```iecst
(*Destinations*)

TYPE
	SystemDestinationsEnum :
		(
		DEST_STARTUP,
		DEST_PROCESS_1 := 10,
		DEST_PROCESS_1A,
		DEST_PROCESS_1B,
		DEST_PROCESS_2 := 20,
		DEST_PROCESS_2A,
		DEST_PROCESS_2B,
		DEST_PROCESS_3 := 30
		);
	SystemDestinationsTyp : 	STRUCT
		Name : STRING[32];
		Sector : McSectorType;
		Position : LREAL;
	END_STRUCT;
END_TYPE
```

Listed in the project but not available here: Logical/Source/Main/Exit.st, Logical/Source/Main/Types.typ, Logical/Source/Main/Variables.var
